LIN {X -0.158,Y -301.655,Z 469.672,A 0.000,B 0.000,C 90.000,E1 301.003} C_DIS
LIN {X -0.099,Y -317.062,Z 469.654,A 0.000,B 0.000,C 90.000,E1 297.719} C_DIS
LIN {X -0.042,Y -330.950,Z 469.640,A 0.000,B 0.000,C 90.000,E1 295.155} C_DIS
LIN {X 0.084,Y -344.129,Z 469.628,A 0.000,B 0.000,C 90.000,E1 292.950} C_DIS
LIN {X -0.112,Y -362.871,Z 469.612,A 0.000,B 0.000,C 90.000,E1 290.248} C_DIS
LIN {X -0.023,Y -381.291,Z 469.599,A 0.000,B 0.000,C 90.000,E1 287.873} C_DIS
LIN {X 0.019,Y -403.542,Z 469.585,A 0.000,B 0.000,C 90.000,E1 285.300} C_DIS
LIN {X 0.221,Y -426.591,Z 469.572,A 0.000,B 0.000,C 90.000,E1 282.883} C_DIS
LIN {X 0.019,Y -436.659,Z 469.566,A 0.000,B 0.000,C 90.000,E1 281.883} C_DIS
LIN {X 0.090,Y -446.267,Z 469.560,A 0.000,B 0.000,C 90.000,E1 280.838} C_DIS
LIN {X 0.109,Y -455.363,Z 469.554,A 0.000,B 0.000,C 90.000,E1 279.792} C_DIS
LIN {X 0.000,Y -461.575,Z 469.550,A 0.000,B 0.000,C 90.000,E1 279.029} C_DIS
LIN {X -0.130,Y -467.256,Z 469.546,A 0.000,B 0.000,C 90.000,E1 278.276} C_DIS
LIN {X 0.187,Y -472.386,Z 469.542,A 0.000,B 0.000,C 90.000,E1 277.473} C_DIS
LIN {X 0.155,Y -476.926,Z 469.537,A 0.000,B 0.000,C 90.000,E1 276.720} C_DIS
LIN {X 0.153,Y -480.963,Z 469.533,A 0.000,B 0.000,C 90.000,E1 275.967} C_DIS
LIN {X 0.136,Y -484.414,Z 469.529,A 0.000,B 0.000,C 90.000,E1 275.220} C_DIS
LIN {X 0.150,Y -487.205,Z 469.525,A 0.000,B 0.000,C 90.000,E1 274.473} C_DIS
LIN {X -0.144,Y -488.693,Z 469.522,A 0.000,B 0.000,C 90.000,E1 274.012} C_DIS
LIN {X 0.025,Y -489.834,Z 469.519,A 0.000,B 0.000,C 90.000,E1 273.498} C_DIS
LIN {X 0.235,Y -490.624,Z 469.517,A 0.000,B 0.000,C 90.000,E1 272.980} C_DIS
LIN {X -0.066,Y -491.068,Z 469.514,A 0.000,B 0.000,C 90.000,E1 272.522} C_DIS
LIN {X 0.131,Y -491.117,Z 469.511,A 0.000,B 0.000,C 90.000,E1 272.007} C_DIS
LIN {X -0.143,Y -490.735,Z 469.509,A 0.000,B 0.000,C 90.000,E1 271.547} C_DIS
LIN {X 0.057,Y -489.896,Z 469.506,A 0.000,B 0.000,C 90.000,E1 271.031} C_DIS
LIN {X -0.233,Y -488.534,Z 469.503,A 0.000,B 0.000,C 90.000,E1 270.573} C_DIS
LIN {X -0.038,Y -486.619,Z 469.500,A 0.000,B 0.000,C 90.000,E1 270.057} C_DIS
LIN {X 0.147,Y -484.034,Z 469.498,A 0.000,B 0.000,C 90.000,E1 269.542} C_DIS
LIN {X -0.168,Y -480.744,Z 469.495,A 0.000,B 0.000,C 90.000,E1 269.083} C_DIS
LIN {X -0.020,Y -476.512,Z 469.492,A 0.000,B 0.000,C 90.000,E1 268.568} C_DIS
LIN {X 0.119,Y -471.190,Z 469.489,A 0.000,B 0.000,C 90.000,E1 268.051} C_DIS
LIN {X 0.111,Y -465.151,Z 469.487,A 0.000,B 0.000,C 90.000,E1 267.593} C_DIS
LIN {X 0.111,Y -458.674,Z 469.484,A 0.000,B 0.000,C 90.000,E1 267.192} C_DIS
LIN {X 0.149,Y -452.078,Z 469.483,A 0.000,B 0.000,C 90.000,E1 266.849} C_DIS
LIN {X 0.109,Y -444.919,Z 469.481,A 0.000,B 0.000,C 90.000,E1 266.560} C_DIS
LIN {X 0.022,Y -437.347,Z 469.480,A 0.000,B 0.000,C 90.000,E1 266.331} C_DIS
LIN {X -0.069,Y -429.037,Z 469.479,A 0.000,B 0.000,C 90.000,E1 266.159} C_DIS
LIN {X -0.159,Y -419.638,Z 469.478,A 0.000,B 0.000,C 90.000,E1 266.045} C_DIS
LIN {X 0.136,Y -408.844,Z 469.477,A 0.000,B 0.000,C 90.000,E1 265.927} C_DIS
LIN {X 0.025,Y -180.917,Z 469.477,A 0.000,B 0.000,C 90.000,E1 265.927} C_DIS
LIN {X 0.054,Y -180.840,Z 469.472,A 0.000,B 0.000,C 90.000,E1 264.894} C_DIS
LIN {X -0.049,Y -178.880,Z 469.443,A 0.000,B 0.000,C 90.000,E1 259.690} C_DIS
LIN {X 0.027,Y -175.923,Z 469.414,A 0.000,B 0.000,C 90.000,E1 254.574} C_DIS
LIN {X -0.027,Y -175.360,Z 469.410,A 0.000,B 0.000,C 90.000,E1 253.740} C_DIS
LIN {X 0.031,Y -172.139,Z 469.386,A 0.000,B 0.000,C 90.000,E1 249.444} C_DIS
LIN {X 0.009,Y -171.602,Z 469.381,A 0.000,B 0.000,C 90.000,E1 248.592} C_DIS
LIN {X -0.003,Y -167.826,Z 469.357,A 0.000,B 0.000,C 90.000,E1 244.280} C_DIS
LIN {X 0.014,Y -166.550,Z 469.347,A 0.000,B 0.000,C 90.000,E1 242.538} C_DIS
LIN {X -0.074,Y -162.546,Z 469.323,A 0.000,B 0.000,C 90.000,E1 238.201} C_DIS
LIN {X -0.015,Y -161.223,Z 469.313,A 0.000,B 0.000,C 90.000,E1 236.421} C_DIS
LIN {X 0.021,Y -157.230,Z 469.289,A 0.000,B 0.000,C 90.000,E1 231.984} C_DIS
LIN {X 0.044,Y -155.955,Z 469.279,A 0.000,B 0.000,C 90.000,E1 230.194} C_DIS
LIN {X 0.002,Y -152.208,Z 469.254,A 0.000,B 0.000,C 90.000,E1 225.729} C_DIS
LIN {X 0.023,Y -150.452,Z 469.239,A 0.000,B 0.000,C 90.000,E1 223.014} C_DIS
LIN {X 0.050,Y -147.178,Z 469.214,A 0.000,B 0.000,C 90.000,E1 218.463} C_DIS
LIN {X 0.017,Y -145.195,Z 469.193,A 0.000,B 0.000,C 90.000,E1 214.818} C_DIS
LIN {X 0.051,Y -142.335,Z 469.163,A 0.000,B 0.000,C 90.000,E1 209.283} C_DIS
LIN {X -0.020,Y -141.724,Z 469.153,A 0.000,B 0.000,C 90.000,E1 207.462} C_DIS
LIN {X -0.038,Y -139.479,Z 469.116,A 0.000,B 0.000,C 90.000,E1 200.972} C_DIS
LIN {X -0.048,Y -138.976,Z 469.101,A 0.000,B 0.000,C 90.000,E1 198.181} C_DIS
LIN {X 0.073,Y -138.332,Z 469.054,A 0.000,B 0.000,C 90.000,E1 189.726} C_DIS
LIN {X -0.063,Y -139.432,Z 469.008,A 0.000,B 0.000,C 90.000,E1 181.375} C_DIS
LIN {X 0.017,Y -140.957,Z 468.976,A 0.000,B 0.000,C 90.000,E1 175.755} C_DIS
LIN {X -0.033,Y -142.713,Z 468.956,A 0.000,B 0.000,C 90.000,E1 172.064} C_DIS
LIN {X 0.067,Y -145.090,Z 468.930,A 0.000,B 0.000,C 90.000,E1 167.409} C_DIS
LIN {X 0.061,Y -147.714,Z 468.910,A 0.000,B 0.000,C 90.000,E1 163.740} C_DIS
LIN {X 0.003,Y -150.372,Z 468.890,A 0.000,B 0.000,C 90.000,E1 160.115} C_DIS
LIN {X 0.021,Y -153.799,Z 468.869,A 0.000,B 0.000,C 90.000,E1 156.485} C_DIS
LIN {X 0.081,Y -157.211,Z 468.849,A 0.000,B 0.000,C 90.000,E1 152.871} C_DIS
LIN {X 0.022,Y -161.376,Z 468.830,A 0.000,B 0.000,C 90.000,E1 149.331} C_DIS
LIN {X 0.033,Y -165.578,Z 468.810,A 0.000,B 0.000,C 90.000,E1 145.801} C_DIS
LIN {X 0.020,Y -170.497,Z 468.791,A 0.000,B 0.000,C 90.000,E1 142.316} C_DIS
LIN {X 0.065,Y -175.378,Z 468.772,A 0.000,B 0.000,C 90.000,E1 138.852} C_DIS
LIN {X -0.073,Y -181.002,Z 468.753,A 0.000,B 0.000,C 90.000,E1 135.486} C_DIS
LIN {X 0.051,Y -186.430,Z 468.734,A 0.000,B 0.000,C 90.000,E1 132.081} C_DIS
LIN {X 0.121,Y -191.056,Z 468.720,A 0.000,B 0.000,C 90.000,E1 129.564} C_DIS
LIN {X -0.048,Y -194.103,Z 468.710,A 0.000,B 0.000,C 90.000,E1 127.810} C_DIS
LIN {X -0.108,Y -291.699,Z 468.710,A 0.000,B 0.000,C 90.000,E1 127.810} C_DIS
LIN {X 0.063,Y -294.118,Z 468.710,A 0.000,B 0.000,C 90.000,E1 127.729} C_DIS
LIN {X -0.041,Y -299.359,Z 468.708,A 0.000,B 0.000,C 90.000,E1 127.443} C_DIS
LIN {X -0.149,Y -302.223,Z 468.706,A 0.000,B 0.000,C 90.000,E1 127.156} C_DIS
LIN {X 0.030,Y -304.266,Z 468.705,A 0.000,B 0.000,C 90.000,E1 126.824} C_DIS
LIN {X 0.149,Y -305.872,Z 468.703,A 0.000,B 0.000,C 90.000,E1 126.503} C_DIS
LIN {X -0.076,Y -307.278,Z 468.701,A 0.000,B 0.000,C 90.000,E1 126.217} C_DIS
LIN {X -0.055,Y -310.333,Z 468.696,A 0.000,B 0.000,C 90.000,E1 125.231} C_DIS
LIN {X -0.088,Y -320.951,Z 468.678,A 0.000,B 0.000,C 90.000,E1 122.005} C_DIS
LIN {X -0.112,Y -331.871,Z 468.662,A 0.000,B 0.000,C 90.000,E1 119.155} C_DIS
LIN {X -0.150,Y -344.193,Z 468.646,A 0.000,B 0.000,C 90.000,E1 116.360} C_DIS
LIN {X -0.016,Y -356.409,Z 468.633,A 0.000,B 0.000,C 90.000,E1 113.898} C_DIS
LIN {X -0.187,Y -369.906,Z 468.619,A 0.000,B 0.000,C 90.000,E1 111.535} C_DIS
LIN {X 0.190,Y -384.783,Z 468.607,A 0.000,B 0.000,C 90.000,E1 109.141} C_DIS
LIN {X -0.174,Y -401.147,Z 468.594,A 0.000,B 0.000,C 90.000,E1 106.913} C_DIS
LIN {X 0.022,Y -419.122,Z 468.581,A 0.000,B 0.000,C 90.000,E1 104.662} C_DIS
LIN {X -0.150,Y -438.706,Z 468.570,A 0.000,B 0.000,C 90.000,E1 102.535} C_DIS
LIN {X -0.130,Y -459.049,Z 468.559,A 0.000,B 0.000,C 90.000,E1 100.546} C_DIS
LIN {X -0.157,Y -482.472,Z 468.547,A 0.000,B 0.000,C 90.000,E1 98.511} C_DIS
LIN {X 0.005,Y -484.489,Z 468.546,A 0.000,B 0.000,C 90.000,E1 98.276} C_DIS
LIN {X -0.183,Y -486.247,Z 468.545,A 0.000,B 0.000,C 90.000,E1 98.049} C_DIS
LIN {X 0.181,Y -487.565,Z 468.543,A 0.000,B 0.000,C 90.000,E1 97.757} C_DIS
LIN {X -0.103,Y -489.207,Z 468.540,A 0.000,B 0.000,C 90.000,E1 97.296} C_DIS
LIN {X 0.106,Y -489.773,Z 468.538,A 0.000,B 0.000,C 90.000,E1 96.777} C_DIS
LIN {X -0.163,Y -489.358,Z 468.535,A 0.000,B 0.000,C 90.000,E1 96.315} C_DIS
LIN {X 0.059,Y -487.894,Z 468.532,A 0.000,B 0.000,C 90.000,E1 95.796} C_DIS
LIN {X -0.099,Y -486.692,Z 468.531,A 0.000,B 0.000,C 90.000,E1 95.568} C_DIS
LIN {X -0.209,Y -485.083,Z 468.530,A 0.000,B 0.000,C 90.000,E1 95.334} C_DIS
LIN {X -0.049,Y -475.019,Z 468.523,A 0.000,B 0.000,C 90.000,E1 94.073} C_DIS
LIN {X 0.111,Y -457.545,Z 468.510,A 0.000,B 0.000,C 90.000,E1 91.776} C_DIS
LIN {X -0.163,Y -445.267,Z 468.500,A 0.000,B 0.000,C 90.000,E1 90.000} C_DIS
LIN {X -0.208,Y -433.697,Z 468.490,A 0.000,B 0.000,C 90.000,E1 88.165} C_DIS
LIN {X 0.193,Y -419.113,Z 468.476,A 0.000,B 0.000,C 90.000,E1 85.698} C_DIS
LIN {X 0.149,Y -406.464,Z 468.464,A 0.000,B 0.000,C 90.000,E1 83.514} C_DIS
LIN {X -0.112,Y -395.623,Z 468.453,A 0.000,B 0.000,C 90.000,E1 81.602} C_DIS
LIN {X -0.159,Y -383.212,Z 468.441,A 0.000,B 0.000,C 90.000,E1 79.342} C_DIS
LIN {X 0.080,Y -369.445,Z 468.426,A 0.000,B 0.000,C 90.000,E1 76.700} C_DIS
LIN {X 0.029,Y -356.550,Z 468.411,A 0.000,B 0.000,C 90.000,E1 74.047} C_DIS
LIN {X 0.030,Y -345.025,Z 468.396,A 0.000,B 0.000,C 90.000,E1 71.329} C_DIS
LIN {X -0.159,Y -333.470,Z 468.379,A 0.000,B 0.000,C 90.000,E1 68.284} C_DIS
LIN {X 0.056,Y -324.572,Z 468.365,A 0.000,B 0.000,C 90.000,E1 65.741} C_DIS
LIN {X 0.091,Y -316.945,Z 468.353,A 0.000,B 0.000,C 90.000,E1 63.512} C_DIS
LIN {X -0.098,Y -308.433,Z 468.339,A 0.000,B 0.000,C 90.000,E1 60.973} C_DIS
LIN {X 0.074,Y -300.074,Z 468.324,A 0.000,B 0.000,C 90.000,E1 58.329} C_DIS
LIN {X 0.002,Y -290.135,Z 468.306,A 0.000,B 0.000,C 90.000,E1 55.022} C_DIS
LIN {X 0.033,Y -282.648,Z 468.291,A 0.000,B 0.000,C 90.000,E1 52.316} C_DIS
LIN {X -0.008,Y -276.960,Z 468.279,A 0.000,B 0.000,C 90.000,E1 50.275} C_DIS
LIN {X 0.010,Y -270.921,Z 468.268,A 0.000,B 0.000,C 90.000,E1 48.200} C_DIS
LIN {X -0.127,Y -264.601,Z 468.256,A 0.000,B 0.000,C 90.000,E1 46.134} C_DIS
LIN {X 0.179,Y -258.110,Z 468.244,A 0.000,B 0.000,C 90.000,E1 43.947} C_DIS
LIN {X 0.002,Y -251.544,Z 468.232,A 0.000,B 0.000,C 90.000,E1 41.838} C_DIS
LIN {X 0.090,Y -242.873,Z 468.216,A 0.000,B 0.000,C 90.000,E1 38.910} C_DIS
LIN {X 0.041,Y -234.668,Z 468.200,A 0.000,B 0.000,C 90.000,E1 35.964} C_DIS
LIN {X 0.033,Y -227.225,Z 468.183,A 0.000,B 0.000,C 90.000,E1 32.959} C_DIS
LIN {X -0.030,Y -220.513,Z 468.166,A 0.000,B 0.000,C 90.000,E1 29.922} C_DIS
LIN {X -0.007,Y -214.701,Z 468.149,A 0.000,B 0.000,C 90.000,E1 26.821} C_DIS
LIN {X 0.001,Y -208.464,Z 468.127,A 0.000,B 0.000,C 90.000,E1 22.898} C_DIS
LIN {X 0.067,Y -203.248,Z 468.105,A 0.000,B 0.000,C 90.000,E1 18.906} C_DIS
LIN {X 0.035,Y -199.029,Z 468.083,A 0.000,B 0.000,C 90.000,E1 14.898} C_DIS
LIN {X 0.082,Y -195.313,Z 468.056,A 0.000,B 0.000,C 90.000,E1 10.018} C_DIS
LIN {X 0.005,Y -192.428,Z 468.019,A 0.000,B 0.000,C 90.000,E1 3.498} C_DIS
LIN {X 0.027,Y -193.612,Z 467.956,A 0.000,B 0.000,C 90.000,E1 352.129} C_DIS
LIN {X 0.005,Y -196.608,Z 467.929,A 0.000,B 0.000,C 90.000,E1 347.229} C_DIS
LIN {X -0.008,Y -200.943,Z 467.902,A 0.000,B 0.000,C 90.000,E1 342.362} C_DIS
LIN {X 0.006,Y -205.588,Z 467.880,A 0.000,B 0.000,C 90.000,E1 338.337} C_DIS
LIN {X 0.009,Y -211.093,Z 467.858,A 0.000,B 0.000,C 90.000,E1 334.357} C_DIS
LIN {X 0.119,Y -216.069,Z 467.840,A 0.000,B 0.000,C 90.000,E1 331.179} C_DIS
LIN {X -0.017,Y -222.825,Z 467.818,A 0.000,B 0.000,C 90.000,E1 327.327} C_DIS
LIN {X -0.029,Y -230.159,Z 467.797,A 0.000,B 0.000,C 90.000,E1 323.497} C_DIS
LIN {X 0.053,Y -238.285,Z 467.776,A 0.000,B 0.000,C 90.000,E1 319.703} C_DIS
LIN {X -0.003,Y -245.579,Z 467.760,A 0.000,B 0.000,C 90.000,E1 316.743} C_DIS
LIN {X -0.036,Y -254.769,Z 467.741,A 0.000,B 0.000,C 90.000,E1 313.461} C_DIS
LIN {X -0.120,Y -265.095,Z 467.723,A 0.000,B 0.000,C 90.000,E1 310.253} C_DIS
LIN {X -0.037,Y -276.415,Z 467.706,A 0.000,B 0.000,C 90.000,E1 307.076} C_DIS
LIN {X -0.074,Y -288.634,Z 467.689,A 0.000,B 0.000,C 90.000,E1 303.992} C_DIS
LIN {X 0.173,Y -301.649,Z 467.672,A 0.000,B 0.000,C 90.000,E1 300.924} C_DIS
LIN {X -0.037,Y -317.088,Z 467.654,A 0.000,B 0.000,C 90.000,E1 297.692} C_DIS
LIN {X -0.065,Y -334.625,Z 467.636,A 0.000,B 0.000,C 90.000,E1 294.515} C_DIS
LIN {X -0.003,Y -346.171,Z 467.626,A 0.000,B 0.000,C 90.000,E1 292.642} C_DIS
LIN {X -0.208,Y -362.890,Z 467.612,A 0.000,B 0.000,C 90.000,E1 290.248} C_DIS
LIN {X -0.127,Y -383.715,Z 467.598,A 0.000,B 0.000,C 90.000,E1 287.583} C_DIS
LIN {X 0.056,Y -406.100,Z 467.583,A 0.000,B 0.000,C 90.000,E1 285.009} C_DIS
LIN {X 0.110,Y -426.722,Z 467.572,A 0.000,B 0.000,C 90.000,E1 282.883} C_DIS
LIN {X -0.120,Y -436.847,Z 467.566,A 0.000,B 0.000,C 90.000,E1 281.883} C_DIS
LIN {X -0.146,Y -446.582,Z 467.560,A 0.000,B 0.000,C 90.000,E1 280.838} C_DIS
LIN {X 0.116,Y -453.506,Z 467.556,A 0.000,B 0.000,C 90.000,E1 280.018} C_DIS
LIN {X 0.189,Y -461.868,Z 467.550,A 0.000,B 0.000,C 90.000,E1 278.973} C_DIS
LIN {X 0.065,Y -467.543,Z 467.546,A 0.000,B 0.000,C 90.000,E1 278.219} C_DIS
LIN {X -0.018,Y -472.658,Z 467.541,A 0.000,B 0.000,C 90.000,E1 277.466} C_DIS
LIN {X -0.111,Y -477.174,Z 467.537,A 0.000,B 0.000,C 90.000,E1 276.720} C_DIS
LIN {X -0.115,Y -481.179,Z 467.533,A 0.000,B 0.000,C 90.000,E1 275.967} C_DIS
LIN {X -0.130,Y -484.631,Z 467.529,A 0.000,B 0.000,C 90.000,E1 275.220} C_DIS
LIN {X -0.116,Y -487.443,Z 467.525,A 0.000,B 0.000,C 90.000,E1 274.473} C_DIS
LIN {X 0.077,Y -488.925,Z 467.522,A 0.000,B 0.000,C 90.000,E1 273.955} C_DIS
LIN {X -0.240,Y -490.031,Z 467.519,A 0.000,B 0.000,C 90.000,E1 273.498} C_DIS
LIN {X -0.029,Y -490.816,Z 467.517,A 0.000,B 0.000,C 90.000,E1 272.980} C_DIS
LIN {X 0.161,Y -491.229,Z 467.514,A 0.000,B 0.000,C 90.000,E1 272.465} C_DIS
LIN {X -0.131,Y -491.240,Z 467.511,A 0.000,B 0.000,C 90.000,E1 272.007} C_DIS
LIN {X 0.085,Y -490.808,Z 467.508,A 0.000,B 0.000,C 90.000,E1 271.489} C_DIS
LIN {X -0.203,Y -489.908,Z 467.506,A 0.000,B 0.000,C 90.000,E1 271.031} C_DIS
LIN {X -0.004,Y -488.535,Z 467.503,A 0.000,B 0.000,C 90.000,E1 270.516} C_DIS
LIN {X 0.190,Y -486.545,Z 467.500,A 0.000,B 0.000,C 90.000,E1 270.000} C_DIS
LIN {X -0.109,Y -483.920,Z 467.497,A 0.000,B 0.000,C 90.000,E1 269.542} C_DIS
LIN {X 0.057,Y -480.586,Z 467.495,A 0.000,B 0.000,C 90.000,E1 269.026} C_DIS
LIN {X 0.203,Y -476.308,Z 467.492,A 0.000,B 0.000,C 90.000,E1 268.511} C_DIS
LIN {X -0.133,Y -470.890,Z 467.489,A 0.000,B 0.000,C 90.000,E1 268.051} C_DIS
LIN {X -0.113,Y -464.803,Z 467.487,A 0.000,B 0.000,C 90.000,E1 267.593} C_DIS
LIN {X -0.072,Y -458.342,Z 467.484,A 0.000,B 0.000,C 90.000,E1 267.192} C_DIS
LIN {X 0.019,Y -451.643,Z 467.482,A 0.000,B 0.000,C 90.000,E1 266.846} C_DIS
LIN {X 0.058,Y -444.877,Z 467.481,A 0.000,B 0.000,C 90.000,E1 266.560} C_DIS
LIN {X -0.068,Y -437.009,Z 467.480,A 0.000,B 0.000,C 90.000,E1 266.331} C_DIS
LIN {X -0.150,Y -428.528,Z 467.479,A 0.000,B 0.000,C 90.000,E1 266.159} C_DIS
LIN {X -0.216,Y -418.896,Z 467.478,A 0.000,B 0.000,C 90.000,E1 266.045} C_DIS
LIN {X 0.111,Y -408.269,Z 467.477,A 0.000,B 0.000,C 90.000,E1 265.927} C_DIS
LIN {X 0.016,Y -180.917,Z 467.477,A 0.000,B 0.000,C 90.000,E1 265.927} C_DIS
LIN {X 0.047,Y -180.838,Z 467.472,A 0.000,B 0.000,C 90.000,E1 264.894} C_DIS
LIN {X -0.055,Y -178.879,Z 467.443,A 0.000,B 0.000,C 90.000,E1 259.690} C_DIS
LIN {X 0.020,Y -175.922,Z 467.414,A 0.000,B 0.000,C 90.000,E1 254.574} C_DIS
LIN {X -0.090,Y -174.620,Z 467.405,A 0.000,B 0.000,C 90.000,E1 252.906} C_DIS
LIN {X 0.002,Y -171.601,Z 467.381,A 0.000,B 0.000,C 90.000,E1 248.592} C_DIS
LIN {X -0.009,Y -167.823,Z 467.357,A 0.000,B 0.000,C 90.000,E1 244.280} C_DIS
LIN {X 0.008,Y -166.548,Z 467.347,A 0.000,B 0.000,C 90.000,E1 242.538} C_DIS
LIN {X -0.081,Y -162.544,Z 467.323,A 0.000,B 0.000,C 90.000,E1 238.201} C_DIS
LIN {X -0.021,Y -161.221,Z 467.313,A 0.000,B 0.000,C 90.000,E1 236.421} C_DIS
LIN {X 0.014,Y -157.228,Z 467.289,A 0.000,B 0.000,C 90.000,E1 231.984} C_DIS
LIN {X 0.037,Y -155.953,Z 467.279,A 0.000,B 0.000,C 90.000,E1 230.194} C_DIS
LIN {X -0.004,Y -152.206,Z 467.254,A 0.000,B 0.000,C 90.000,E1 225.729} C_DIS
LIN {X 0.016,Y -150.451,Z 467.239,A 0.000,B 0.000,C 90.000,E1 223.014} C_DIS
LIN {X 0.043,Y -147.177,Z 467.214,A 0.000,B 0.000,C 90.000,E1 218.463} C_DIS
LIN {X 0.010,Y -145.195,Z 467.193,A 0.000,B 0.000,C 90.000,E1 214.818} C_DIS
LIN {X 0.045,Y -142.334,Z 467.163,A 0.000,B 0.000,C 90.000,E1 209.283} C_DIS
LIN {X -0.026,Y -141.723,Z 467.152,A 0.000,B 0.000,C 90.000,E1 207.462} C_DIS
LIN {X -0.044,Y -139.478,Z 467.116,A 0.000,B 0.000,C 90.000,E1 200.972} C_DIS
LIN {X -0.055,Y -138.976,Z 467.101,A 0.000,B 0.000,C 90.000,E1 198.181} C_DIS
LIN {X 0.067,Y -138.332,Z 467.054,A 0.000,B 0.000,C 90.000,E1 189.726} C_DIS
LIN {X 0.070,Y -139.431,Z 467.007,A 0.000,B 0.000,C 90.000,E1 181.318} C_DIS
LIN {X 0.010,Y -140.958,Z 466.976,A 0.000,B 0.000,C 90.000,E1 175.755} C_DIS
LIN {X -0.040,Y -142.714,Z 466.956,A 0.000,B 0.000,C 90.000,E1 172.064} C_DIS
LIN {X 0.060,Y -145.091,Z 466.930,A 0.000,B 0.000,C 90.000,E1 167.409} C_DIS
LIN {X 0.056,Y -147.716,Z 466.910,A 0.000,B 0.000,C 90.000,E1 163.740} C_DIS
LIN {X -0.004,Y -150.373,Z 466.890,A 0.000,B 0.000,C 90.000,E1 160.115} C_DIS
LIN {X 0.014,Y -153.802,Z 466.869,A 0.000,B 0.000,C 90.000,E1 156.485} C_DIS
LIN {X 0.074,Y -157.213,Z 466.849,A 0.000,B 0.000,C 90.000,E1 152.871} C_DIS
LIN {X 0.015,Y -161.378,Z 466.830,A 0.000,B 0.000,C 90.000,E1 149.331} C_DIS
LIN {X 0.027,Y -165.581,Z 466.810,A 0.000,B 0.000,C 90.000,E1 145.801} C_DIS
LIN {X 0.013,Y -170.501,Z 466.791,A 0.000,B 0.000,C 90.000,E1 142.316} C_DIS
LIN {X 0.058,Y -175.381,Z 466.772,A 0.000,B 0.000,C 90.000,E1 138.852} C_DIS
LIN {X -0.080,Y -181.006,Z 466.753,A 0.000,B 0.000,C 90.000,E1 135.486} C_DIS
LIN {X 0.044,Y -186.434,Z 466.734,A 0.000,B 0.000,C 90.000,E1 132.081} C_DIS
LIN {X 0.113,Y -191.060,Z 466.720,A 0.000,B 0.000,C 90.000,E1 129.564} C_DIS
LIN {X 0.032,Y -194.204,Z 466.710,A 0.000,B 0.000,C 90.000,E1 127.729} C_DIS
LIN {X 0.014,Y -291.917,Z 466.710,A 0.000,B 0.000,C 90.000,E1 127.729} C_DIS
LIN {X 0.121,Y -294.651,Z 466.709,A 0.000,B 0.000,C 90.000,E1 127.649} C_DIS
LIN {X 0.010,Y -299.269,Z 466.708,A 0.000,B 0.000,C 90.000,E1 127.397} C_DIS
LIN {X -0.160,Y -301.942,Z 466.706,A 0.000,B 0.000,C 90.000,E1 127.156} C_DIS
LIN {X -0.180,Y -305.655,Z 466.703,A 0.000,B 0.000,C 90.000,E1 126.583} C_DIS
LIN {X 0.016,Y -307.140,Z 466.701,A 0.000,B 0.000,C 90.000,E1 126.217} C_DIS
LIN {X 0.034,Y -308.314,Z 466.699,A 0.000,B 0.000,C 90.000,E1 125.884} C_DIS
LIN {X 0.119,Y -318.630,Z 466.681,A 0.000,B 0.000,C 90.000,E1 122.625} C_DIS
LIN {X -0.083,Y -329.246,Z 466.665,A 0.000,B 0.000,C 90.000,E1 119.795} C_DIS
LIN {X 0.103,Y -341.240,Z 466.650,A 0.000,B 0.000,C 90.000,E1 116.950} C_DIS
LIN {X 0.036,Y -354.714,Z 466.635,A 0.000,B 0.000,C 90.000,E1 114.207} C_DIS
LIN {X -0.176,Y -368.038,Z 466.621,A 0.000,B 0.000,C 90.000,E1 111.844} C_DIS
LIN {X 0.153,Y -382.727,Z 466.608,A 0.000,B 0.000,C 90.000,E1 109.450} C_DIS
LIN {X 0.124,Y -398.891,Z 466.595,A 0.000,B 0.000,C 90.000,E1 107.166} C_DIS
LIN {X -0.008,Y -416.646,Z 466.583,A 0.000,B 0.000,C 90.000,E1 104.954} C_DIS
LIN {X 0.138,Y -436.049,Z 466.571,A 0.000,B 0.000,C 90.000,E1 102.771} C_DIS
LIN {X -0.010,Y -456.318,Z 466.560,A 0.000,B 0.000,C 90.000,E1 100.782} C_DIS
LIN {X 0.184,Y -477.118,Z 466.550,A 0.000,B 0.000,C 90.000,E1 98.916} C_DIS
LIN {X -0.077,Y -482.359,Z 466.547,A 0.000,B 0.000,C 90.000,E1 98.511} C_DIS
LIN {X 0.084,Y -484.444,Z 466.546,A 0.000,B 0.000,C 90.000,E1 98.276} C_DIS
LIN {X -0.103,Y -486.255,Z 466.545,A 0.000,B 0.000,C 90.000,E1 98.049} C_DIS
LIN {X -0.223,Y -487.615,Z 466.543,A 0.000,B 0.000,C 90.000,E1 97.814} C_DIS
LIN {X -0.024,Y -489.315,Z 466.541,A 0.000,B 0.000,C 90.000,E1 97.296} C_DIS
LIN {X 0.186,Y -489.931,Z 466.538,A 0.000,B 0.000,C 90.000,E1 96.777} C_DIS
LIN {X -0.083,Y -489.561,Z 466.535,A 0.000,B 0.000,C 90.000,E1 96.315} C_DIS
LIN {X 0.140,Y -488.153,Z 466.532,A 0.000,B 0.000,C 90.000,E1 95.796} C_DIS
LIN {X -0.018,Y -486.984,Z 466.531,A 0.000,B 0.000,C 90.000,E1 95.568} C_DIS
LIN {X -0.127,Y -485.420,Z 466.530,A 0.000,B 0.000,C 90.000,E1 95.334} C_DIS
LIN {X 0.036,Y -475.390,Z 466.523,A 0.000,B 0.000,C 90.000,E1 94.073} C_DIS
LIN {X -0.021,Y -456.050,Z 466.509,A 0.000,B 0.000,C 90.000,E1 91.547} C_DIS
LIN {X -0.123,Y -442.244,Z 466.497,A 0.000,B 0.000,C 90.000,E1 89.484} C_DIS
LIN {X 0.057,Y -427.435,Z 466.484,A 0.000,B 0.000,C 90.000,E1 87.078} C_DIS
LIN {X -0.116,Y -413.042,Z 466.470,A 0.000,B 0.000,C 90.000,E1 84.666} C_DIS
LIN {X 0.194,Y -400.568,Z 466.458,A 0.000,B 0.000,C 90.000,E1 82.413} C_DIS
LIN {X -0.178,Y -389.678,Z 466.447,A 0.000,B 0.000,C 90.000,E1 80.500} C_DIS
LIN {X 0.024,Y -380.432,Z 466.438,A 0.000,B 0.000,C 90.000,E1 78.757} C_DIS
LIN {X -0.189,Y -365.347,Z 466.421,A 0.000,B 0.000,C 90.000,E1 75.880} C_DIS
LIN {X -0.195,Y -354.196,Z 466.408,A 0.000,B 0.000,C 90.000,E1 73.504} C_DIS
LIN {X 0.080,Y -342.919,Z 466.393,A 0.000,B 0.000,C 90.000,E1 70.732} C_DIS
LIN {X -0.060,Y -331.475,Z 466.376,A 0.000,B 0.000,C 90.000,E1 67.667} C_DIS
LIN {X -0.109,Y -321.458,Z 466.360,A 0.000,B 0.000,C 90.000,E1 64.845} C_DIS
LIN {X -0.071,Y -312.772,Z 466.346,A 0.000,B 0.000,C 90.000,E1 62.281} C_DIS
LIN {X 0.060,Y -304.280,Z 466.332,A 0.000,B 0.000,C 90.000,E1 59.665} C_DIS
LIN {X 0.038,Y -294.052,Z 466.313,A 0.000,B 0.000,C 90.000,E1 56.373} C_DIS
LIN {X -0.127,Y -284.513,Z 466.295,A 0.000,B 0.000,C 90.000,E1 53.050} C_DIS
LIN {X 0.086,Y -278.881,Z 466.283,A 0.000,B 0.000,C 90.000,E1 50.964} C_DIS
LIN {X -0.069,Y -272.948,Z 466.272,A 0.000,B 0.000,C 90.000,E1 48.933} C_DIS
LIN {X 0.032,Y -266.721,Z 466.260,A 0.000,B 0.000,C 90.000,E1 46.824} C_DIS
LIN {X 0.010,Y -260.324,Z 466.248,A 0.000,B 0.000,C 90.000,E1 44.717} C_DIS
LIN {X -0.127,Y -253.782,Z 466.237,A 0.000,B 0.000,C 90.000,E1 42.609} C_DIS
LIN {X 0.000,Y -247.246,Z 466.225,A 0.000,B 0.000,C 90.000,E1 40.415} C_DIS
LIN {X -0.008,Y -236.714,Z 466.204,A 0.000,B 0.000,C 90.000,E1 36.744} C_DIS
LIN {X -0.152,Y -229.104,Z 466.188,A 0.000,B 0.000,C 90.000,E1 33.785} C_DIS
LIN {X -0.045,Y -222.146,Z 466.171,A 0.000,B 0.000,C 90.000,E1 30.718} C_DIS
LIN {X -0.073,Y -216.122,Z 466.153,A 0.000,B 0.000,C 90.000,E1 27.641} C_DIS
LIN {X -0.063,Y -210.880,Z 466.136,A 0.000,B 0.000,C 90.000,E1 24.515} C_DIS
LIN {X -0.039,Y -205.232,Z 466.114,A 0.000,B 0.000,C 90.000,E1 20.556} C_DIS
LIN {X -0.021,Y -200.601,Z 466.092,A 0.000,B 0.000,C 90.000,E1 16.551} C_DIS
LIN {X -0.100,Y -196.945,Z 466.069,A 0.000,B 0.000,C 90.000,E1 12.535} C_DIS
LIN {X 0.084,Y -193.512,Z 466.038,A 0.000,B 0.000,C 90.000,E1 6.777} C_DIS
LIN {X 0.080,Y -193.113,Z 465.961,A 0.000,B 0.000,C 90.000,E1 352.932} C_DIS
LIN {X -0.006,Y -196.481,Z 465.929,A 0.000,B 0.000,C 90.000,E1 347.229} C_DIS
LIN {X -0.025,Y -200.783,Z 465.902,A 0.000,B 0.000,C 90.000,E1 342.362} C_DIS
LIN {X -0.017,Y -205.404,Z 465.880,A 0.000,B 0.000,C 90.000,E1 338.337} C_DIS
LIN {X 0.071,Y -210.921,Z 465.858,A 0.000,B 0.000,C 90.000,E1 334.332} C_DIS
LIN {X 0.030,Y -217.220,Z 465.836,A 0.000,B 0.000,C 90.000,E1 330.411} C_DIS
LIN {X -0.058,Y -222.680,Z 465.818,A 0.000,B 0.000,C 90.000,E1 327.327} C_DIS
LIN {X -0.075,Y -229.999,Z 465.797,A 0.000,B 0.000,C 90.000,E1 323.497} C_DIS
LIN {X 0.000,Y -238.139,Z 465.776,A 0.000,B 0.000,C 90.000,E1 319.703} C_DIS
LIN {X 0.084,Y -247.370,Z 465.756,A 0.000,B 0.000,C 90.000,E1 315.972} C_DIS
LIN {X 0.122,Y -256.853,Z 465.737,A 0.000,B 0.000,C 90.000,E1 312.690} C_DIS
LIN {X 0.105,Y -267.433,Z 465.719,A 0.000,B 0.000,C 90.000,E1 309.483} C_DIS
LIN {X -0.078,Y -279.034,Z 465.702,A 0.000,B 0.000,C 90.000,E1 306.377} C_DIS
LIN {X -0.055,Y -292.877,Z 465.683,A 0.000,B 0.000,C 90.000,E1 302.959} C_DIS
LIN {X 0.000,Y -306.143,Z 465.666,A 0.000,B 0.000,C 90.000,E1 299.951} C_DIS
LIN {X 0.146,Y -320.455,Z 465.650,A 0.000,B 0.000,C 90.000,E1 297.001} C_DIS
LIN {X -0.063,Y -338.348,Z 465.633,A 0.000,B 0.000,C 90.000,E1 293.875} C_DIS
LIN {X 0.018,Y -356.478,Z 465.617,A 0.000,B 0.000,C 90.000,E1 291.099} C_DIS
LIN {X -0.101,Y -369.646,Z 465.607,A 0.000,B 0.000,C 90.000,E1 289.322} C_DIS
LIN {X 0.095,Y -393.537,Z 465.591,A 0.000,B 0.000,C 90.000,E1 286.386} C_DIS
LIN {X -0.102,Y -416.450,Z 465.577,A 0.000,B 0.000,C 90.000,E1 283.939} C_DIS
LIN {X 0.189,Y -431.864,Z 465.569,A 0.000,B 0.000,C 90.000,E1 282.355} C_DIS
LIN {X -0.156,Y -441.778,Z 465.563,A 0.000,B 0.000,C 90.000,E1 281.366} C_DIS
LIN {X -0.109,Y -451.273,Z 465.557,A 0.000,B 0.000,C 90.000,E1 280.310} C_DIS
LIN {X -0.065,Y -459.852,Z 465.551,A 0.000,B 0.000,C 90.000,E1 279.265} C_DIS
LIN {X -0.213,Y -465.749,Z 465.547,A 0.000,B 0.000,C 90.000,E1 278.511} C_DIS
LIN {X 0.159,Y -471.043,Z 465.543,A 0.000,B 0.000,C 90.000,E1 277.701} C_DIS
LIN {X 0.107,Y -475.760,Z 465.539,A 0.000,B 0.000,C 90.000,E1 276.947} C_DIS
LIN {X 0.044,Y -479.960,Z 465.534,A 0.000,B 0.000,C 90.000,E1 276.201} C_DIS
LIN {X 0.019,Y -483.618,Z 465.530,A 0.000,B 0.000,C 90.000,E1 275.454} C_DIS
LIN {X 0.197,Y -485.745,Z 465.528,A 0.000,B 0.000,C 90.000,E1 274.935} C_DIS
LIN {X -0.097,Y -487.565,Z 465.525,A 0.000,B 0.000,C 90.000,E1 274.473} C_DIS
LIN {X 0.098,Y -489.058,Z 465.522,A 0.000,B 0.000,C 90.000,E1 273.955} C_DIS
LIN {X -0.219,Y -490.199,Z 465.519,A 0.000,B 0.000,C 90.000,E1 273.498} C_DIS
LIN {X -0.008,Y -490.973,Z 465.517,A 0.000,B 0.000,C 90.000,E1 272.980} C_DIS
LIN {X 0.185,Y -491.371,Z 465.514,A 0.000,B 0.000,C 90.000,E1 272.465} C_DIS
LIN {X -0.107,Y -491.331,Z 465.511,A 0.000,B 0.000,C 90.000,E1 272.007} C_DIS
LIN {X 0.110,Y -490.932,Z 465.508,A 0.000,B 0.000,C 90.000,E1 271.489} C_DIS
LIN {X -0.178,Y -490.012,Z 465.506,A 0.000,B 0.000,C 90.000,E1 271.031} C_DIS
LIN {X 0.023,Y -488.622,Z 465.503,A 0.000,B 0.000,C 90.000,E1 270.516} C_DIS
LIN {X 0.217,Y -486.643,Z 465.500,A 0.000,B 0.000,C 90.000,E1 270.000} C_DIS
LIN {X -0.083,Y -484.046,Z 465.497,A 0.000,B 0.000,C 90.000,E1 269.542} C_DIS
LIN {X -0.240,Y -482.489,Z 465.496,A 0.000,B 0.000,C 90.000,E1 269.312} C_DIS
LIN {X -0.082,Y -478.649,Z 465.493,A 0.000,B 0.000,C 90.000,E1 268.797} C_DIS
LIN {X 0.231,Y -476.420,Z 465.492,A 0.000,B 0.000,C 90.000,E1 268.511} C_DIS
LIN {X -0.105,Y -471.016,Z 465.489,A 0.000,B 0.000,C 90.000,E1 268.051} C_DIS
LIN {X -0.100,Y -464.953,Z 465.487,A 0.000,B 0.000,C 90.000,E1 267.593} C_DIS
LIN {X -0.071,Y -458.484,Z 465.484,A 0.000,B 0.000,C 90.000,E1 267.192} C_DIS
LIN {X -0.021,Y -451.645,Z 465.482,A 0.000,B 0.000,C 90.000,E1 266.846} C_DIS
LIN {X 0.012,Y -444.807,Z 465.481,A 0.000,B 0.000,C 90.000,E1 266.560} C_DIS
LIN {X -0.088,Y -437.088,Z 465.480,A 0.000,B 0.000,C 90.000,E1 266.331} C_DIS
LIN {X -0.166,Y -428.532,Z 465.479,A 0.000,B 0.000,C 90.000,E1 266.159} C_DIS
LIN {X 0.187,Y -418.720,Z 465.478,A 0.000,B 0.000,C 90.000,E1 265.988} C_DIS
LIN {X 0.104,Y -407.968,Z 465.477,A 0.000,B 0.000,C 90.000,E1 265.927} C_DIS
LIN {X 0.013,Y -180.917,Z 465.477,A 0.000,B 0.000,C 90.000,E1 265.927} C_DIS
LIN {X 0.045,Y -180.839,Z 465.472,A 0.000,B 0.000,C 90.000,E1 264.894} C_DIS
LIN {X -0.058,Y -178.879,Z 465.443,A 0.000,B 0.000,C 90.000,E1 259.690} C_DIS
LIN {X 0.018,Y -175.922,Z 465.414,A 0.000,B 0.000,C 90.000,E1 254.574} C_DIS
LIN {X -0.093,Y -174.619,Z 465.405,A 0.000,B 0.000,C 90.000,E1 252.906} C_DIS
LIN {X 0.000,Y -171.600,Z 465.381,A 0.000,B 0.000,C 90.000,E1 248.592} C_DIS
LIN {X -0.012,Y -167.823,Z 465.357,A 0.000,B 0.000,C 90.000,E1 244.280} C_DIS
LIN {X 0.006,Y -166.547,Z 465.347,A 0.000,B 0.000,C 90.000,E1 242.538} C_DIS
LIN {X -0.083,Y -162.543,Z 465.323,A 0.000,B 0.000,C 90.000,E1 238.201} C_DIS
LIN {X -0.023,Y -161.221,Z 465.313,A 0.000,B 0.000,C 90.000,E1 236.421} C_DIS
LIN {X 0.012,Y -157.227,Z 465.289,A 0.000,B 0.000,C 90.000,E1 231.984} C_DIS
LIN {X 0.035,Y -155.952,Z 465.279,A 0.000,B 0.000,C 90.000,E1 230.194} C_DIS
LIN {X -0.006,Y -152.205,Z 465.254,A 0.000,B 0.000,C 90.000,E1 225.729} C_DIS
LIN {X 0.015,Y -150.451,Z 465.239,A 0.000,B 0.000,C 90.000,E1 223.014} C_DIS
LIN {X 0.041,Y -147.176,Z 465.214,A 0.000,B 0.000,C 90.000,E1 218.463} C_DIS
LIN {X 0.009,Y -145.193,Z 465.193,A 0.000,B 0.000,C 90.000,E1 214.818} C_DIS
LIN {X 0.043,Y -142.334,Z 465.163,A 0.000,B 0.000,C 90.000,E1 209.283} C_DIS
LIN {X -0.028,Y -141.723,Z 465.152,A 0.000,B 0.000,C 90.000,E1 207.462} C_DIS
LIN {X -0.045,Y -139.478,Z 465.116,A 0.000,B 0.000,C 90.000,E1 200.972} C_DIS
LIN {X -0.057,Y -138.976,Z 465.101,A 0.000,B 0.000,C 90.000,E1 198.181} C_DIS
LIN {X 0.065,Y -138.331,Z 465.054,A 0.000,B 0.000,C 90.000,E1 189.726} C_DIS
LIN {X 0.068,Y -139.431,Z 465.007,A 0.000,B 0.000,C 90.000,E1 181.318} C_DIS
LIN {X 0.008,Y -140.958,Z 464.976,A 0.000,B 0.000,C 90.000,E1 175.755} C_DIS
LIN {X -0.042,Y -142.714,Z 464.956,A 0.000,B 0.000,C 90.000,E1 172.064} C_DIS
LIN {X 0.058,Y -145.092,Z 464.930,A 0.000,B 0.000,C 90.000,E1 167.409} C_DIS
LIN {X 0.054,Y -147.717,Z 464.910,A 0.000,B 0.000,C 90.000,E1 163.740} C_DIS
LIN {X -0.006,Y -150.374,Z 464.890,A 0.000,B 0.000,C 90.000,E1 160.115} C_DIS
LIN {X 0.013,Y -153.803,Z 464.869,A 0.000,B 0.000,C 90.000,E1 156.485} C_DIS
LIN {X 0.072,Y -157.214,Z 464.849,A 0.000,B 0.000,C 90.000,E1 152.871} C_DIS
LIN {X 0.013,Y -161.380,Z 464.830,A 0.000,B 0.000,C 90.000,E1 149.331} C_DIS
LIN {X 0.024,Y -165.582,Z 464.810,A 0.000,B 0.000,C 90.000,E1 145.801} C_DIS
LIN {X 0.010,Y -170.502,Z 464.791,A 0.000,B 0.000,C 90.000,E1 142.316} C_DIS
LIN {X 0.055,Y -175.383,Z 464.771,A 0.000,B 0.000,C 90.000,E1 138.852} C_DIS
LIN {X -0.082,Y -181.007,Z 464.753,A 0.000,B 0.000,C 90.000,E1 135.486} C_DIS
LIN {X 0.042,Y -186.435,Z 464.734,A 0.000,B 0.000,C 90.000,E1 132.081} C_DIS
LIN {X 0.111,Y -191.061,Z 464.720,A 0.000,B 0.000,C 90.000,E1 129.564} C_DIS
LIN {X 0.023,Y -194.290,Z 464.709,A 0.000,B 0.000,C 90.000,E1 127.684} C_DIS
LIN {X -0.015,Y -291.952,Z 464.709,A 0.000,B 0.000,C 90.000,E1 127.684} C_DIS
LIN {X 0.114,Y -292.785,Z 464.709,A 0.000,B 0.000,C 90.000,E1 127.649} C_DIS
LIN {X 0.005,Y -298.761,Z 464.708,A 0.000,B 0.000,C 90.000,E1 127.397} C_DIS
LIN {X -0.164,Y -301.629,Z 464.706,A 0.000,B 0.000,C 90.000,E1 127.156} C_DIS
LIN {X -0.018,Y -305.348,Z 464.703,A 0.000,B 0.000,C 90.000,E1 126.583} C_DIS
LIN {X -0.003,Y -306.929,Z 464.701,A 0.000,B 0.000,C 90.000,E1 126.251} C_DIS
LIN {X -0.055,Y -308.179,Z 464.700,A 0.000,B 0.000,C 90.000,E1 125.931} C_DIS
LIN {X 0.086,Y -319.620,Z 464.680,A 0.000,B 0.000,C 90.000,E1 122.339} C_DIS
LIN {X 0.024,Y -330.373,Z 464.664,A 0.000,B 0.000,C 90.000,E1 119.489} C_DIS
LIN {X -0.043,Y -342.509,Z 464.648,A 0.000,B 0.000,C 90.000,E1 116.693} C_DIS
LIN {X -0.086,Y -356.143,Z 464.633,A 0.000,B 0.000,C 90.000,E1 113.951} C_DIS
LIN {X 0.073,Y -369.617,Z 464.620,A 0.000,B 0.000,C 90.000,E1 111.535} C_DIS
LIN {X -0.038,Y -384.469,Z 464.607,A 0.000,B 0.000,C 90.000,E1 109.214} C_DIS
LIN {X 0.091,Y -400.807,Z 464.594,A 0.000,B 0.000,C 90.000,E1 106.913} C_DIS
LIN {X -0.115,Y -418.752,Z 464.582,A 0.000,B 0.000,C 90.000,E1 104.717} C_DIS
LIN {X 0.114,Y -438.316,Z 464.570,A 0.000,B 0.000,C 90.000,E1 102.535} C_DIS
LIN {X 0.121,Y -458.650,Z 464.559,A 0.000,B 0.000,C 90.000,E1 100.546} C_DIS
LIN {X 0.080,Y -482.125,Z 464.547,A 0.000,B 0.000,C 90.000,E1 98.511} C_DIS
LIN {X 0.241,Y -484.310,Z 464.546,A 0.000,B 0.000,C 90.000,E1 98.276} C_DIS
LIN {X 0.105,Y -486.155,Z 464.545,A 0.000,B 0.000,C 90.000,E1 98.049} C_DIS
LIN {X 0.037,Y -487.549,Z 464.543,A 0.000,B 0.000,C 90.000,E1 97.814} C_DIS
LIN {X 0.236,Y -489.362,Z 464.541,A 0.000,B 0.000,C 90.000,E1 97.296} C_DIS
LIN {X -0.041,Y -490.070,Z 464.538,A 0.000,B 0.000,C 90.000,E1 96.834} C_DIS
LIN {X 0.178,Y -489.791,Z 464.535,A 0.000,B 0.000,C 90.000,E1 96.315} C_DIS
LIN {X -0.086,Y -488.485,Z 464.532,A 0.000,B 0.000,C 90.000,E1 95.853} C_DIS
LIN {X -0.242,Y -487.380,Z 464.531,A 0.000,B 0.000,C 90.000,E1 95.625} C_DIS
LIN {X 0.133,Y -485.896,Z 464.530,A 0.000,B 0.000,C 90.000,E1 95.334} C_DIS
LIN {X -0.002,Y -477.985,Z 464.524,A 0.000,B 0.000,C 90.000,E1 94.359} C_DIS
LIN {X -0.005,Y -458.402,Z 464.510,A 0.000,B 0.000,C 90.000,E1 91.835} C_DIS
LIN {X 0.200,Y -446.025,Z 464.500,A 0.000,B 0.000,C 90.000,E1 90.000} C_DIS
LIN {X -0.116,Y -432.740,Z 464.488,A 0.000,B 0.000,C 90.000,E1 87.936} C_DIS
LIN {X -0.160,Y -418.208,Z 464.475,A 0.000,B 0.000,C 90.000,E1 85.527} C_DIS
LIN {X -0.120,Y -404.092,Z 464.461,A 0.000,B 0.000,C 90.000,E1 83.053} C_DIS
LIN {X -0.032,Y -393.230,Z 464.450,A 0.000,B 0.000,C 90.000,E1 81.084} C_DIS
LIN {X -0.110,Y -382.444,Z 464.439,A 0.000,B 0.000,C 90.000,E1 79.106} C_DIS
LIN {X 0.102,Y -367.262,Z 464.423,A 0.000,B 0.000,C 90.000,E1 76.172} C_DIS
LIN {X 0.136,Y -355.964,Z 464.410,A 0.000,B 0.000,C 90.000,E1 73.795} C_DIS
LIN {X 0.024,Y -344.501,Z 464.395,A 0.000,B 0.000,C 90.000,E1 71.094} C_DIS
LIN {X -0.064,Y -332.916,Z 464.378,A 0.000,B 0.000,C 90.000,E1 68.028} C_DIS
LIN {X 0.136,Y -323.925,Z 464.364,A 0.000,B 0.000,C 90.000,E1 65.485} C_DIS
LIN {X 0.076,Y -315.172,Z 464.350,A 0.000,B 0.000,C 90.000,E1 62.948} C_DIS
LIN {X -0.026,Y -306.578,Z 464.335,A 0.000,B 0.000,C 90.000,E1 60.383} C_DIS
LIN {X -0.125,Y -296.182,Z 464.317,A 0.000,B 0.000,C 90.000,E1 57.120} C_DIS
LIN {X 0.015,Y -286.475,Z 464.299,A 0.000,B 0.000,C 90.000,E1 53.749} C_DIS
LIN {X 0.095,Y -280.864,Z 464.287,A 0.000,B 0.000,C 90.000,E1 51.698} C_DIS
LIN {X -0.024,Y -275.032,Z 464.276,A 0.000,B 0.000,C 90.000,E1 49.666} C_DIS
LIN {X 0.138,Y -268.910,Z 464.264,A 0.000,B 0.000,C 90.000,E1 47.553} C_DIS
LIN {X -0.034,Y -262.614,Z 464.253,A 0.000,B 0.000,C 90.000,E1 45.486} C_DIS
LIN {X 0.053,Y -256.120,Z 464.241,A 0.000,B 0.000,C 90.000,E1 43.338} C_DIS
LIN {X -0.153,Y -249.593,Z 464.229,A 0.000,B 0.000,C 90.000,E1 41.229} C_DIS
LIN {X 0.063,Y -238.917,Z 464.209,A 0.000,B 0.000,C 90.000,E1 37.523} C_DIS
LIN {X 0.101,Y -231.073,Z 464.192,A 0.000,B 0.000,C 90.000,E1 34.532} C_DIS
LIN {X -0.060,Y -223.930,Z 464.175,A 0.000,B 0.000,C 90.000,E1 31.544} C_DIS
LIN {X 0.069,Y -217.631,Z 464.158,A 0.000,B 0.000,C 90.000,E1 28.437} C_DIS
LIN {X 0.022,Y -212.219,Z 464.141,A 0.000,B 0.000,C 90.000,E1 25.335} C_DIS
LIN {X -0.032,Y -206.343,Z 464.119,A 0.000,B 0.000,C 90.000,E1 21.408} C_DIS
LIN {X 0.022,Y -201.480,Z 464.097,A 0.000,B 0.000,C 90.000,E1 17.402} C_DIS
LIN {X 0.074,Y -197.604,Z 464.074,A 0.000,B 0.000,C 90.000,E1 13.355} C_DIS
LIN {X -0.050,Y -194.288,Z 464.047,A 0.000,B 0.000,C 90.000,E1 8.511} C_DIS
LIN {X -0.030,Y -191.907,Z 464.011,A 0.000,B 0.000,C 90.000,E1 1.949} C_DIS
LIN {X 0.014,Y -193.359,Z 463.956,A 0.000,B 0.000,C 90.000,E1 352.129} C_DIS
LIN {X -0.018,Y -196.344,Z 463.929,A 0.000,B 0.000,C 90.000,E1 347.229} C_DIS
LIN {X 0.063,Y -199.825,Z 463.906,A 0.000,B 0.000,C 90.000,E1 343.142} C_DIS
LIN {X -0.027,Y -204.225,Z 463.884,A 0.000,B 0.000,C 90.000,E1 339.135} C_DIS
LIN {X -0.060,Y -209.574,Z 463.862,A 0.000,B 0.000,C 90.000,E1 335.153} C_DIS
LIN {X 0.051,Y -215.741,Z 463.840,A 0.000,B 0.000,C 90.000,E1 331.179} C_DIS
LIN {X 0.007,Y -221.136,Z 463.823,A 0.000,B 0.000,C 90.000,E1 328.074} C_DIS
LIN {X 0.132,Y -228.335,Z 463.801,A 0.000,B 0.000,C 90.000,E1 324.196} C_DIS
LIN {X 0.017,Y -236.269,Z 463.780,A 0.000,B 0.000,C 90.000,E1 320.436} C_DIS
LIN {X 0.059,Y -245.287,Z 463.760,A 0.000,B 0.000,C 90.000,E1 316.701} C_DIS
LIN {X 0.026,Y -254.523,Z 463.741,A 0.000,B 0.000,C 90.000,E1 313.419} C_DIS
LIN {X 0.120,Y -264.911,Z 463.723,A 0.000,B 0.000,C 90.000,E1 310.172} C_DIS
LIN {X 0.038,Y -276.307,Z 463.706,A 0.000,B 0.000,C 90.000,E1 307.030} C_DIS
LIN {X 0.044,Y -287.168,Z 463.690,A 0.000,B 0.000,C 90.000,E1 304.278} C_DIS
LIN {X -0.001,Y -300.170,Z 463.674,A 0.000,B 0.000,C 90.000,E1 301.258} C_DIS
LIN {X 0.013,Y -315.546,Z 463.655,A 0.000,B 0.000,C 90.000,E1 297.975} C_DIS
LIN {X -0.004,Y -325.701,Z 463.645,A 0.000,B 0.000,C 90.000,E1 296.052} C_DIS
LIN {X 0.132,Y -342.225,Z 463.629,A 0.000,B 0.000,C 90.000,E1 293.206} C_DIS
LIN {X 0.069,Y -362.928,Z 463.612,A 0.000,B 0.000,C 90.000,E1 290.174} C_DIS
LIN {X -0.187,Y -386.207,Z 463.596,A 0.000,B 0.000,C 90.000,E1 287.275} C_DIS
LIN {X -0.068,Y -406.081,Z 463.583,A 0.000,B 0.000,C 90.000,E1 285.009} C_DIS
LIN {X -0.072,Y -426.388,Z 463.572,A 0.000,B 0.000,C 90.000,E1 282.939} C_DIS
LIN {X 0.067,Y -436.511,Z 463.566,A 0.000,B 0.000,C 90.000,E1 281.895} C_DIS
LIN {X 0.156,Y -446.287,Z 463.560,A 0.000,B 0.000,C 90.000,E1 280.838} C_DIS
LIN {X -0.027,Y -453.225,Z 463.556,A 0.000,B 0.000,C 90.000,E1 280.074} C_DIS
LIN {X 0.040,Y -461.635,Z 463.550,A 0.000,B 0.000,C 90.000,E1 279.029} C_DIS
LIN {X -0.089,Y -467.364,Z 463.546,A 0.000,B 0.000,C 90.000,E1 278.276} C_DIS
LIN {X -0.239,Y -472.504,Z 463.542,A 0.000,B 0.000,C 90.000,E1 277.530} C_DIS
LIN {X 0.200,Y -477.056,Z 463.537,A 0.000,B 0.000,C 90.000,E1 276.720} C_DIS
LIN {X 0.198,Y -481.115,Z 463.533,A 0.000,B 0.000,C 90.000,E1 275.967} C_DIS
LIN {X 0.184,Y -484.683,Z 463.529,A 0.000,B 0.000,C 90.000,E1 275.220} C_DIS
LIN {X 0.200,Y -487.583,Z 463.525,A 0.000,B 0.000,C 90.000,E1 274.473} C_DIS
LIN {X -0.092,Y -489.110,Z 463.522,A 0.000,B 0.000,C 90.000,E1 274.012} C_DIS
LIN {X 0.079,Y -490.290,Z 463.519,A 0.000,B 0.000,C 90.000,E1 273.498} C_DIS
LIN {X -0.199,Y -491.079,Z 463.517,A 0.000,B 0.000,C 90.000,E1 273.037} C_DIS
LIN {X -0.007,Y -491.501,Z 463.514,A 0.000,B 0.000,C 90.000,E1 272.522} C_DIS
LIN {X 0.193,Y -491.460,Z 463.511,A 0.000,B 0.000,C 90.000,E1 272.007} C_DIS
LIN {X -0.079,Y -491.084,Z 463.509,A 0.000,B 0.000,C 90.000,E1 271.547} C_DIS
LIN {X 0.122,Y -490.175,Z 463.506,A 0.000,B 0.000,C 90.000,E1 271.031} C_DIS
LIN {X -0.166,Y -488.804,Z 463.503,A 0.000,B 0.000,C 90.000,E1 270.573} C_DIS
LIN {X 0.031,Y -486.898,Z 463.500,A 0.000,B 0.000,C 90.000,E1 270.057} C_DIS
LIN {X 0.218,Y -484.347,Z 463.498,A 0.000,B 0.000,C 90.000,E1 269.542} C_DIS
LIN {X -0.097,Y -481.063,Z 463.495,A 0.000,B 0.000,C 90.000,E1 269.083} C_DIS
LIN {X 0.053,Y -476.822,Z 463.492,A 0.000,B 0.000,C 90.000,E1 268.568} C_DIS
LIN {X 0.192,Y -471.543,Z 463.489,A 0.000,B 0.000,C 90.000,E1 268.051} C_DIS
LIN {X 0.162,Y -465.574,Z 463.487,A 0.000,B 0.000,C 90.000,E1 267.593} C_DIS
LIN {X 0.091,Y -458.949,Z 463.484,A 0.000,B 0.000,C 90.000,E1 267.192} C_DIS
LIN {X 0.124,Y -452.271,Z 463.483,A 0.000,B 0.000,C 90.000,E1 266.849} C_DIS
LIN {X 0.129,Y -445.261,Z 463.481,A 0.000,B 0.000,C 90.000,E1 266.560} C_DIS
LIN {X 0.029,Y -437.817,Z 463.480,A 0.000,B 0.000,C 90.000,E1 266.331} C_DIS
LIN {X -0.058,Y -429.417,Z 463.479,A 0.000,B 0.000,C 90.000,E1 266.159} C_DIS
LIN {X -0.136,Y -420.085,Z 463.478,A 0.000,B 0.000,C 90.000,E1 266.045} C_DIS
LIN {X 0.101,Y -407.405,Z 463.477,A 0.000,B 0.000,C 90.000,E1 265.927} C_DIS
LIN {X 0.022,Y -180.917,Z 463.477,A 0.000,B 0.000,C 90.000,E1 265.927} C_DIS
LIN {X -0.075,Y -180.871,Z 463.472,A 0.000,B 0.000,C 90.000,E1 265.065} C_DIS
LIN {X -0.018,Y -178.986,Z 463.444,A 0.000,B 0.000,C 90.000,E1 259.982} C_DIS
LIN {X -0.007,Y -177.966,Z 463.435,A 0.000,B 0.000,C 90.000,E1 258.285} C_DIS
LIN {X 0.012,Y -175.608,Z 463.411,A 0.000,B 0.000,C 90.000,E1 254.031} C_DIS
LIN {X 0.024,Y -172.332,Z 463.388,A 0.000,B 0.000,C 90.000,E1 249.752} C_DIS
LIN {X 0.003,Y -171.808,Z 463.383,A 0.000,B 0.000,C 90.000,E1 248.901} C_DIS
LIN {X 0.011,Y -170.269,Z 463.373,A 0.000,B 0.000,C 90.000,E1 247.177} C_DIS
LIN {X -0.053,Y -166.811,Z 463.349,A 0.000,B 0.000,C 90.000,E1 242.871} C_DIS
LIN {X 0.004,Y -162.793,Z 463.325,A 0.000,B 0.000,C 90.000,E1 238.486} C_DIS
LIN {X 0.064,Y -161.481,Z 463.315,A 0.000,B 0.000,C 90.000,E1 236.707} C_DIS
LIN {X -0.020,Y -157.477,Z 463.291,A 0.000,B 0.000,C 90.000,E1 232.316} C_DIS
LIN {X 0.037,Y -155.492,Z 463.276,A 0.000,B 0.000,C 90.000,E1 229.622} C_DIS
LIN {X -0.031,Y -151.798,Z 463.251,A 0.000,B 0.000,C 90.000,E1 225.162} C_DIS
LIN {X -0.017,Y -150.007,Z 463.236,A 0.000,B 0.000,C 90.000,E1 222.447} C_DIS
LIN {X 0.014,Y -146.834,Z 463.211,A 0.000,B 0.000,C 90.000,E1 217.890} C_DIS
LIN {X 0.000,Y -145.415,Z 463.195,A 0.000,B 0.000,C 90.000,E1 215.152} C_DIS
LIN {X 0.036,Y -142.844,Z 463.170,A 0.000,B 0.000,C 90.000,E1 210.541} C_DIS
LIN {X -0.035,Y -141.458,Z 463.149,A 0.000,B 0.000,C 90.000,E1 206.873} C_DIS
LIN {X 0.005,Y -139.374,Z 463.113,A 0.000,B 0.000,C 90.000,E1 200.355} C_DIS
LIN {X -0.053,Y -138.824,Z 463.098,A 0.000,B 0.000,C 90.000,E1 197.583} C_DIS
LIN {X 0.036,Y -138.352,Z 463.056,A 0.000,B 0.000,C 90.000,E1 190.074} C_DIS
LIN {X 0.009,Y -139.531,Z 463.004,A 0.000,B 0.000,C 90.000,E1 180.745} C_DIS
LIN {X -0.038,Y -141.212,Z 462.973,A 0.000,B 0.000,C 90.000,E1 175.179} C_DIS
LIN {X 0.062,Y -142.586,Z 462.958,A 0.000,B 0.000,C 90.000,E1 172.356} C_DIS
LIN {X 0.016,Y -144.884,Z 462.932,A 0.000,B 0.000,C 90.000,E1 167.757} C_DIS
LIN {X -0.030,Y -147.510,Z 462.912,A 0.000,B 0.000,C 90.000,E1 164.102} C_DIS
LIN {X 0.045,Y -150.104,Z 462.891,A 0.000,B 0.000,C 90.000,E1 160.423} C_DIS
LIN {X 0.056,Y -153.461,Z 462.871,A 0.000,B 0.000,C 90.000,E1 156.794} C_DIS
LIN {X -0.091,Y -157.825,Z 462.846,A 0.000,B 0.000,C 90.000,E1 152.359} C_DIS
LIN {X -0.061,Y -162.108,Z 462.827,A 0.000,B 0.000,C 90.000,E1 148.791} C_DIS
LIN {X -0.036,Y -166.309,Z 462.807,A 0.000,B 0.000,C 90.000,E1 145.261} C_DIS
LIN {X 0.066,Y -171.326,Z 462.788,A 0.000,B 0.000,C 90.000,E1 141.743} C_DIS
LIN {X -0.006,Y -176.226,Z 462.768,A 0.000,B 0.000,C 90.000,E1 138.324} C_DIS
LIN {X 0.114,Y -180.506,Z 462.754,A 0.000,B 0.000,C 90.000,E1 135.729} C_DIS
LIN {X 0.094,Y -185.909,Z 462.736,A 0.000,B 0.000,C 90.000,E1 132.366} C_DIS
LIN {X 0.030,Y -190.537,Z 462.722,A 0.000,B 0.000,C 90.000,E1 129.886} C_DIS
LIN {X -0.046,Y -194.389,Z 462.709,A 0.000,B 0.000,C 90.000,E1 127.649} C_DIS
LIN {X -0.109,Y -291.597,Z 462.709,A 0.000,B 0.000,C 90.000,E1 127.649} C_DIS
LIN {X 0.082,Y -292.602,Z 462.709,A 0.000,B 0.000,C 90.000,E1 127.604} C_DIS
LIN {X -0.114,Y -297.798,Z 462.708,A 0.000,B 0.000,C 90.000,E1 127.443} C_DIS
LIN {X 0.126,Y -300.732,Z 462.707,A 0.000,B 0.000,C 90.000,E1 127.156} C_DIS
LIN {X -0.058,Y -304.485,Z 462.704,A 0.000,B 0.000,C 90.000,E1 126.710} C_DIS
LIN {X -0.047,Y -306.288,Z 462.702,A 0.000,B 0.000,C 90.000,E1 126.377} C_DIS
LIN {X 0.146,Y -307.703,Z 462.700,A 0.000,B 0.000,C 90.000,E1 126.011} C_DIS
LIN {X -0.036,Y -311.769,Z 462.693,A 0.000,B 0.000,C 90.000,E1 124.739} C_DIS
LIN {X -0.026,Y -322.619,Z 462.675,A 0.000,B 0.000,C 90.000,E1 121.514} C_DIS
LIN {X -0.172,Y -333.765,Z 462.659,A 0.000,B 0.000,C 90.000,E1 118.693} C_DIS
LIN {X 0.149,Y -346.331,Z 462.644,A 0.000,B 0.000,C 90.000,E1 115.848} C_DIS
LIN {X -0.126,Y -358.780,Z 462.630,A 0.000,B 0.000,C 90.000,E1 113.462} C_DIS
LIN {X 0.105,Y -372.529,Z 462.617,A 0.000,B 0.000,C 90.000,E1 111.046} C_DIS
LIN {X 0.068,Y -387.676,Z 462.604,A 0.000,B 0.000,C 90.000,E1 108.725} C_DIS
LIN {X 0.161,Y -404.334,Z 462.591,A 0.000,B 0.000,C 90.000,E1 106.441} C_DIS
LIN {X 0.051,Y -422.625,Z 462.579,A 0.000,B 0.000,C 90.000,E1 104.245} C_DIS
LIN {X 0.057,Y -442.427,Z 462.567,A 0.000,B 0.000,C 90.000,E1 102.119} C_DIS
LIN {X -0.202,Y -462.874,Z 462.557,A 0.000,B 0.000,C 90.000,E1 100.197} C_DIS
LIN {X -0.150,Y -483.625,Z 462.547,A 0.000,B 0.000,C 90.000,E1 98.398} C_DIS
LIN {X -0.080,Y -485.565,Z 462.545,A 0.000,B 0.000,C 90.000,E1 98.163} C_DIS
LIN {X -0.077,Y -487.049,Z 462.544,A 0.000,B 0.000,C 90.000,E1 97.936} C_DIS
LIN {X -0.188,Y -488.283,Z 462.543,A 0.000,B 0.000,C 90.000,E1 97.701} C_DIS
LIN {X 0.184,Y -489.186,Z 462.541,A 0.000,B 0.000,C 90.000,E1 97.409} C_DIS
LIN {X -0.091,Y -490.153,Z 462.539,A 0.000,B 0.000,C 90.000,E1 96.947} C_DIS
LIN {X 0.127,Y -490.123,Z 462.536,A 0.000,B 0.000,C 90.000,E1 96.429} C_DIS
LIN {X -0.138,Y -489.089,Z 462.533,A 0.000,B 0.000,C 90.000,E1 95.967} C_DIS
LIN {X 0.192,Y -488.147,Z 462.532,A 0.000,B 0.000,C 90.000,E1 95.682} C_DIS
LIN {X 0.037,Y -486.865,Z 462.530,A 0.000,B 0.000,C 90.000,E1 95.454} C_DIS
LIN {X -0.235,Y -483.195,Z 462.528,A 0.000,B 0.000,C 90.000,E1 94.992} C_DIS
LIN {X -0.014,Y -459.509,Z 462.511,A 0.000,B 0.000,C 90.000,E1 91.949} C_DIS
LIN {X 0.213,Y -447.012,Z 462.501,A 0.000,B 0.000,C 90.000,E1 90.115} C_DIS
LIN {X 0.079,Y -432.070,Z 462.488,A 0.000,B 0.000,C 90.000,E1 87.764} C_DIS
LIN {X 0.001,Y -417.530,Z 462.474,A 0.000,B 0.000,C 90.000,E1 85.355} C_DIS
LIN {X 0.068,Y -403.457,Z 462.460,A 0.000,B 0.000,C 90.000,E1 82.875} C_DIS
LIN {X 0.140,Y -392.593,Z 462.450,A 0.000,B 0.000,C 90.000,E1 80.905} C_DIS
LIN {X 0.056,Y -381.816,Z 462.439,A 0.000,B 0.000,C 90.000,E1 78.926} C_DIS
LIN {X -0.106,Y -366.724,Z 462.422,A 0.000,B 0.000,C 90.000,E1 76.047} C_DIS
LIN {X -0.125,Y -356.827,Z 462.411,A 0.000,B 0.000,C 90.000,E1 73.976} C_DIS
LIN {X 0.137,Y -344.061,Z 462.394,A 0.000,B 0.000,C 90.000,E1 70.913} C_DIS
LIN {X 0.030,Y -332.474,Z 462.377,A 0.000,B 0.000,C 90.000,E1 67.847} C_DIS
LIN {X -0.081,Y -323.451,Z 462.363,A 0.000,B 0.000,C 90.000,E1 65.357} C_DIS
LIN {X -0.004,Y -314.656,Z 462.349,A 0.000,B 0.000,C 90.000,E1 62.794} C_DIS
LIN {X -0.032,Y -307.100,Z 462.336,A 0.000,B 0.000,C 90.000,E1 60.539} C_DIS
LIN {X 0.034,Y -296.640,Z 462.318,A 0.000,B 0.000,C 90.000,E1 57.248} C_DIS
LIN {X 0.018,Y -286.866,Z 462.300,A 0.000,B 0.000,C 90.000,E1 53.909} C_DIS
LIN {X -0.119,Y -281.258,Z 462.288,A 0.000,B 0.000,C 90.000,E1 51.904} C_DIS
LIN {X -0.014,Y -275.443,Z 462.277,A 0.000,B 0.000,C 90.000,E1 49.828} C_DIS
LIN {X -0.046,Y -269.344,Z 462.265,A 0.000,B 0.000,C 90.000,E1 47.757} C_DIS
LIN {X -0.011,Y -263.075,Z 462.254,A 0.000,B 0.000,C 90.000,E1 45.648} C_DIS
LIN {X -0.102,Y -256.629,Z 462.242,A 0.000,B 0.000,C 90.000,E1 43.542} C_DIS
LIN {X 0.052,Y -250.108,Z 462.230,A 0.000,B 0.000,C 90.000,E1 41.353} C_DIS
LIN {X -0.068,Y -239.406,Z 462.210,A 0.000,B 0.000,C 90.000,E1 37.729} C_DIS
LIN {X -0.016,Y -231.520,Z 462.193,A 0.000,B 0.000,C 90.000,E1 34.739} C_DIS
LIN {X -0.044,Y -224.333,Z 462.176,A 0.000,B 0.000,C 90.000,E1 31.720} C_DIS
LIN {X 0.087,Y -217.962,Z 462.159,A 0.000,B 0.000,C 90.000,E1 28.615} C_DIS
LIN {X -0.105,Y -211.243,Z 462.137,A 0.000,B 0.000,C 90.000,E1 24.771} C_DIS
LIN {X 0.006,Y -205.505,Z 462.116,A 0.000,B 0.000,C 90.000,E1 20.791} C_DIS
LIN {X -0.030,Y -200.795,Z 462.093,A 0.000,B 0.000,C 90.000,E1 16.804} C_DIS
LIN {X -0.047,Y -197.071,Z 462.071,A 0.000,B 0.000,C 90.000,E1 12.771} C_DIS
LIN {X -0.048,Y -193.465,Z 462.039,A 0.000,B 0.000,C 90.000,E1 7.068} C_DIS
LIN {X 0.070,Y -192.866,Z 461.961,A 0.000,B 0.000,C 90.000,E1 352.932} C_DIS
LIN {X -0.029,Y -196.201,Z 461.929,A 0.000,B 0.000,C 90.000,E1 347.229} C_DIS
LIN {X 0.046,Y -199.678,Z 461.906,A 0.000,B 0.000,C 90.000,E1 343.142} C_DIS
LIN {X -0.048,Y -204.045,Z 461.884,A 0.000,B 0.000,C 90.000,E1 339.135} C_DIS
LIN {X 0.103,Y -209.407,Z 461.862,A 0.000,B 0.000,C 90.000,E1 335.101} C_DIS
LIN {X 0.017,Y -215.585,Z 461.840,A 0.000,B 0.000,C 90.000,E1 331.179} C_DIS
LIN {X -0.031,Y -220.975,Z 461.823,A 0.000,B 0.000,C 90.000,E1 328.074} C_DIS
LIN {X 0.087,Y -228.195,Z 461.801,A 0.000,B 0.000,C 90.000,E1 324.196} C_DIS
LIN {X -0.033,Y -236.121,Z 461.780,A 0.000,B 0.000,C 90.000,E1 320.436} C_DIS
LIN {X 0.002,Y -245.149,Z 461.759,A 0.000,B 0.000,C 90.000,E1 316.701} C_DIS
LIN {X -0.036,Y -254.393,Z 461.741,A 0.000,B 0.000,C 90.000,E1 313.419} C_DIS
LIN {X 0.051,Y -264.813,Z 461.723,A 0.000,B 0.000,C 90.000,E1 310.172} C_DIS
LIN {X -0.035,Y -276.255,Z 461.706,A 0.000,B 0.000,C 90.000,E1 307.030} C_DIS
LIN {X -0.034,Y -287.133,Z 461.690,A 0.000,B 0.000,C 90.000,E1 304.278} C_DIS
LIN {X -0.085,Y -300.161,Z 461.674,A 0.000,B 0.000,C 90.000,E1 301.258} C_DIS
LIN {X -0.074,Y -315.564,Z 461.655,A 0.000,B 0.000,C 90.000,E1 297.975} C_DIS
LIN {X -0.004,Y -327.498,Z 461.643,A 0.000,B 0.000,C 90.000,E1 295.720} C_DIS
LIN {X 0.039,Y -342.266,Z 461.629,A 0.000,B 0.000,C 90.000,E1 293.206} C_DIS
LIN {X -0.029,Y -362.965,Z 461.612,A 0.000,B 0.000,C 90.000,E1 290.174} C_DIS
LIN {X -0.121,Y -388.641,Z 461.594,A 0.000,B 0.000,C 90.000,E1 286.968} C_DIS
LIN {X 0.046,Y -408.620,Z 461.582,A 0.000,B 0.000,C 90.000,E1 284.717} C_DIS
LIN {X 0.021,Y -429.223,Z 461.570,A 0.000,B 0.000,C 90.000,E1 282.647} C_DIS
LIN {X 0.172,Y -439.177,Z 461.565,A 0.000,B 0.000,C 90.000,E1 281.602} C_DIS
LIN {X -0.009,Y -446.513,Z 461.560,A 0.000,B 0.000,C 90.000,E1 280.838} C_DIS
LIN {X -0.016,Y -455.608,Z 461.554,A 0.000,B 0.000,C 90.000,E1 279.792} C_DIS
LIN {X 0.086,Y -463.827,Z 461.549,A 0.000,B 0.000,C 90.000,E1 278.746} C_DIS
LIN {X -0.025,Y -469.341,Z 461.544,A 0.000,B 0.000,C 90.000,E1 277.992} C_DIS
LIN {X -0.085,Y -474.229,Z 461.540,A 0.000,B 0.000,C 90.000,E1 277.239} C_DIS
LIN {X -0.113,Y -478.624,Z 461.536,A 0.000,B 0.000,C 90.000,E1 276.486} C_DIS
LIN {X -0.151,Y -482.569,Z 461.532,A 0.000,B 0.000,C 90.000,E1 275.739} C_DIS
LIN {X -0.156,Y -485.911,Z 461.528,A 0.000,B 0.000,C 90.000,E1 274.992} C_DIS
LIN {X 0.035,Y -487.804,Z 461.525,A 0.000,B 0.000,C 90.000,E1 274.473} C_DIS
LIN {X 0.231,Y -489.311,Z 461.522,A 0.000,B 0.000,C 90.000,E1 273.955} C_DIS
LIN {X -0.084,Y -490.484,Z 461.519,A 0.000,B 0.000,C 90.000,E1 273.498} C_DIS
LIN {X 0.129,Y -491.248,Z 461.517,A 0.000,B 0.000,C 90.000,E1 272.980} C_DIS
LIN {X -0.168,Y -491.627,Z 461.514,A 0.000,B 0.000,C 90.000,E1 272.522} C_DIS
LIN {X 0.033,Y -491.598,Z 461.511,A 0.000,B 0.000,C 90.000,E1 272.007} C_DIS
LIN {X -0.239,Y -491.155,Z 461.508,A 0.000,B 0.000,C 90.000,E1 271.547} C_DIS
LIN {X -0.036,Y -490.237,Z 461.506,A 0.000,B 0.000,C 90.000,E1 271.031} C_DIS
LIN {X 0.166,Y -488.845,Z 461.503,A 0.000,B 0.000,C 90.000,E1 270.516} C_DIS
LIN {X -0.126,Y -486.931,Z 461.500,A 0.000,B 0.000,C 90.000,E1 270.057} C_DIS
LIN {X 0.062,Y -484.336,Z 461.497,A 0.000,B 0.000,C 90.000,E1 269.542} C_DIS
LIN {X 0.229,Y -481.017,Z 461.495,A 0.000,B 0.000,C 90.000,E1 269.026} C_DIS
LIN {X -0.101,Y -476.795,Z 461.492,A 0.000,B 0.000,C 90.000,E1 268.568} C_DIS
LIN {X 0.041,Y -471.462,Z 461.489,A 0.000,B 0.000,C 90.000,E1 268.051} C_DIS
LIN {X 0.023,Y -465.408,Z 461.487,A 0.000,B 0.000,C 90.000,E1 267.593} C_DIS
LIN {X -0.201,Y -462.389,Z 461.486,A 0.000,B 0.000,C 90.000,E1 267.421} C_DIS
LIN {X 0.091,Y -455.844,Z 461.484,A 0.000,B 0.000,C 90.000,E1 267.020} C_DIS
LIN {X -0.070,Y -449.048,Z 461.482,A 0.000,B 0.000,C 90.000,E1 266.731} C_DIS
LIN {X 0.074,Y -441.976,Z 461.480,A 0.000,B 0.000,C 90.000,E1 266.445} C_DIS
LIN {X 0.186,Y -434.065,Z 461.479,A 0.000,B 0.000,C 90.000,E1 266.216} C_DIS
LIN {X -0.117,Y -425.275,Z 461.478,A 0.000,B 0.000,C 90.000,E1 266.102} C_DIS
LIN {X -0.051,Y -415.008,Z 461.478,A 0.000,B 0.000,C 90.000,E1 265.988} C_DIS
LIN {X 0.087,Y -405.845,Z 461.477,A 0.000,B 0.000,C 90.000,E1 265.927} C_DIS
LIN {X 0.017,Y -180.918,Z 461.477,A 0.000,B 0.000,C 90.000,E1 265.927} C_DIS
LIN {X -0.069,Y -180.871,Z 461.472,A 0.000,B 0.000,C 90.000,E1 265.065} C_DIS
LIN {X -0.012,Y -178.987,Z 461.444,A 0.000,B 0.000,C 90.000,E1 259.982} C_DIS
LIN {X 0.000,Y -177.967,Z 461.435,A 0.000,B 0.000,C 90.000,E1 258.285} C_DIS
LIN {X 0.018,Y -175.610,Z 461.411,A 0.000,B 0.000,C 90.000,E1 254.031} C_DIS
LIN {X 0.030,Y -172.333,Z 461.388,A 0.000,B 0.000,C 90.000,E1 249.752} C_DIS
LIN {X 0.009,Y -171.809,Z 461.383,A 0.000,B 0.000,C 90.000,E1 248.901} C_DIS
LIN {X 0.017,Y -170.271,Z 461.373,A 0.000,B 0.000,C 90.000,E1 247.177} C_DIS
LIN {X -0.047,Y -166.812,Z 461.349,A 0.000,B 0.000,C 90.000,E1 242.871} C_DIS
LIN {X 0.010,Y -162.795,Z 461.325,A 0.000,B 0.000,C 90.000,E1 238.486} C_DIS
LIN {X 0.070,Y -161.483,Z 461.315,A 0.000,B 0.000,C 90.000,E1 236.707} C_DIS
LIN {X -0.014,Y -157.478,Z 461.291,A 0.000,B 0.000,C 90.000,E1 232.316} C_DIS
LIN {X 0.043,Y -155.494,Z 461.276,A 0.000,B 0.000,C 90.000,E1 229.622} C_DIS
LIN {X -0.025,Y -151.799,Z 461.251,A 0.000,B 0.000,C 90.000,E1 225.162} C_DIS
LIN {X -0.012,Y -150.009,Z 461.236,A 0.000,B 0.000,C 90.000,E1 222.447} C_DIS
LIN {X 0.020,Y -146.835,Z 461.211,A 0.000,B 0.000,C 90.000,E1 217.890} C_DIS
LIN {X 0.006,Y -145.417,Z 461.195,A 0.000,B 0.000,C 90.000,E1 215.152} C_DIS
LIN {X 0.041,Y -142.845,Z 461.170,A 0.000,B 0.000,C 90.000,E1 210.541} C_DIS
LIN {X -0.028,Y -141.459,Z 461.149,A 0.000,B 0.000,C 90.000,E1 206.873} C_DIS
LIN {X 0.011,Y -139.374,Z 461.113,A 0.000,B 0.000,C 90.000,E1 200.355} C_DIS
LIN {X -0.048,Y -138.825,Z 461.098,A 0.000,B 0.000,C 90.000,E1 197.583} C_DIS
LIN {X 0.041,Y -138.352,Z 461.056,A 0.000,B 0.000,C 90.000,E1 190.074} C_DIS
LIN {X 0.015,Y -139.531,Z 461.004,A 0.000,B 0.000,C 90.000,E1 180.745} C_DIS
LIN {X -0.033,Y -141.210,Z 460.973,A 0.000,B 0.000,C 90.000,E1 175.179} C_DIS
LIN {X 0.068,Y -142.585,Z 460.958,A 0.000,B 0.000,C 90.000,E1 172.356} C_DIS
LIN {X 0.022,Y -144.882,Z 460.932,A 0.000,B 0.000,C 90.000,E1 167.757} C_DIS
LIN {X -0.025,Y -147.509,Z 460.912,A 0.000,B 0.000,C 90.000,E1 164.102} C_DIS
LIN {X 0.050,Y -150.102,Z 460.891,A 0.000,B 0.000,C 90.000,E1 160.423} C_DIS
LIN {X 0.062,Y -153.459,Z 460.871,A 0.000,B 0.000,C 90.000,E1 156.794} C_DIS
LIN {X -0.086,Y -157.822,Z 460.846,A 0.000,B 0.000,C 90.000,E1 152.359} C_DIS
LIN {X -0.054,Y -162.105,Z 460.827,A 0.000,B 0.000,C 90.000,E1 148.791} C_DIS
LIN {X -0.030,Y -166.307,Z 460.807,A 0.000,B 0.000,C 90.000,E1 145.261} C_DIS
LIN {X -0.034,Y -171.323,Z 460.788,A 0.000,B 0.000,C 90.000,E1 141.778} C_DIS
LIN {X 0.000,Y -176.224,Z 460.768,A 0.000,B 0.000,C 90.000,E1 138.324} C_DIS
LIN {X -0.006,Y -180.502,Z 460.754,A 0.000,B 0.000,C 90.000,E1 135.769} C_DIS
LIN {X -0.024,Y -185.906,Z 460.736,A 0.000,B 0.000,C 90.000,E1 132.405} C_DIS
LIN {X 0.036,Y -190.533,Z 460.722,A 0.000,B 0.000,C 90.000,E1 129.886} C_DIS
LIN {X 0.031,Y -194.491,Z 460.709,A 0.000,B 0.000,C 90.000,E1 127.569} C_DIS
LIN {X 0.012,Y -291.941,Z 460.709,A 0.000,B 0.000,C 90.000,E1 127.569} C_DIS
LIN {X -0.104,Y -296.970,Z 460.708,A 0.000,B 0.000,C 90.000,E1 127.443} C_DIS
LIN {X -0.128,Y -299.937,Z 460.707,A 0.000,B 0.000,C 90.000,E1 127.237} C_DIS
LIN {X -0.019,Y -303.680,Z 460.704,A 0.000,B 0.000,C 90.000,E1 126.790} C_DIS
LIN {X 0.087,Y -305.601,Z 460.703,A 0.000,B 0.000,C 90.000,E1 126.457} C_DIS
LIN {X -0.051,Y -307.115,Z 460.701,A 0.000,B 0.000,C 90.000,E1 126.171} C_DIS
LIN {X 0.159,Y -308.380,Z 460.699,A 0.000,B 0.000,C 90.000,E1 125.804} C_DIS
LIN {X 0.048,Y -319.879,Z 460.679,A 0.000,B 0.000,C 90.000,E1 122.260} C_DIS
LIN {X -0.010,Y -330.668,Z 460.663,A 0.000,B 0.000,C 90.000,E1 119.411} C_DIS
LIN {X -0.079,Y -342.849,Z 460.648,A 0.000,B 0.000,C 90.000,E1 116.616} C_DIS
LIN {X 0.021,Y -354.931,Z 460.634,A 0.000,B 0.000,C 90.000,E1 114.155} C_DIS
LIN {X -0.043,Y -368.283,Z 460.621,A 0.000,B 0.000,C 90.000,E1 111.770} C_DIS
LIN {X 0.162,Y -383.004,Z 460.608,A 0.000,B 0.000,C 90.000,E1 109.396} C_DIS
LIN {X -0.119,Y -399.201,Z 460.595,A 0.000,B 0.000,C 90.000,E1 107.149} C_DIS
LIN {X 0.026,Y -416.993,Z 460.583,A 0.000,B 0.000,C 90.000,E1 104.898} C_DIS
LIN {X -0.245,Y -436.443,Z 460.571,A 0.000,B 0.000,C 90.000,E1 102.771} C_DIS
LIN {X 0.153,Y -456.726,Z 460.560,A 0.000,B 0.000,C 90.000,E1 100.715} C_DIS
LIN {X -0.029,Y -480.158,Z 460.548,A 0.000,B 0.000,C 90.000,E1 98.681} C_DIS
LIN {X 0.046,Y -482.785,Z 460.547,A 0.000,B 0.000,C 90.000,E1 98.454} C_DIS
LIN {X 0.193,Y -484.902,Z 460.546,A 0.000,B 0.000,C 90.000,E1 98.219} C_DIS
LIN {X -0.210,Y -486.522,Z 460.545,A 0.000,B 0.000,C 90.000,E1 98.049} C_DIS
LIN {X 0.160,Y -487.934,Z 460.543,A 0.000,B 0.000,C 90.000,E1 97.757} C_DIS
LIN {X -0.017,Y -488.984,Z 460.542,A 0.000,B 0.000,C 90.000,E1 97.530} C_DIS
LIN {X 0.196,Y -490.198,Z 460.539,A 0.000,B 0.000,C 90.000,E1 97.011} C_DIS
LIN {X -0.072,Y -490.392,Z 460.536,A 0.000,B 0.000,C 90.000,E1 96.549} C_DIS
LIN {X 0.154,Y -489.597,Z 460.534,A 0.000,B 0.000,C 90.000,E1 96.030} C_DIS
LIN {X -0.106,Y -487.677,Z 460.531,A 0.000,B 0.000,C 90.000,E1 95.568} C_DIS
LIN {X -0.215,Y -486.175,Z 460.529,A 0.000,B 0.000,C 90.000,E1 95.334} C_DIS
LIN {X 0.136,Y -478.247,Z 460.524,A 0.000,B 0.000,C 90.000,E1 94.302} C_DIS
LIN {X 0.151,Y -458.649,Z 460.510,A 0.000,B 0.000,C 90.000,E1 91.776} C_DIS
LIN {X -0.098,Y -446.235,Z 460.500,A 0.000,B 0.000,C 90.000,E1 90.000} C_DIS
LIN {X 0.184,Y -431.322,Z 460.487,A 0.000,B 0.000,C 90.000,E1 87.593} C_DIS
LIN {X 0.120,Y -416.797,Z 460.473,A 0.000,B 0.000,C 90.000,E1 85.179} C_DIS
LIN {X 0.119,Y -402.747,Z 460.460,A 0.000,B 0.000,C 90.000,E1 82.704} C_DIS
LIN {X 0.107,Y -393.451,Z 460.450,A 0.000,B 0.000,C 90.000,E1 81.027} C_DIS
LIN {X 0.032,Y -382.678,Z 460.439,A 0.000,B 0.000,C 90.000,E1 79.050} C_DIS
LIN {X -0.114,Y -367.585,Z 460.423,A 0.000,B 0.000,C 90.000,E1 76.172} C_DIS
LIN {X -0.066,Y -356.296,Z 460.410,A 0.000,B 0.000,C 90.000,E1 73.795} C_DIS
LIN {X 0.178,Y -343.579,Z 460.393,A 0.000,B 0.000,C 90.000,E1 70.732} C_DIS
LIN {X 0.053,Y -331.968,Z 460.376,A 0.000,B 0.000,C 90.000,E1 67.667} C_DIS
LIN {X 0.010,Y -321.817,Z 460.360,A 0.000,B 0.000,C 90.000,E1 64.845} C_DIS
LIN {X -0.016,Y -314.098,Z 460.348,A 0.000,B 0.000,C 90.000,E1 62.615} C_DIS
LIN {X 0.135,Y -305.427,Z 460.333,A 0.000,B 0.000,C 90.000,E1 59.999} C_DIS
LIN {X 0.121,Y -297.062,Z 460.319,A 0.000,B 0.000,C 90.000,E1 57.375} C_DIS
LIN {X -0.048,Y -287.241,Z 460.300,A 0.000,B 0.000,C 90.000,E1 54.069} C_DIS
LIN {X -0.009,Y -281.600,Z 460.289,A 0.000,B 0.000,C 90.000,E1 52.029} C_DIS
LIN {X -0.071,Y -275.808,Z 460.278,A 0.000,B 0.000,C 90.000,E1 49.989} C_DIS
LIN {X -0.096,Y -269.737,Z 460.266,A 0.000,B 0.000,C 90.000,E1 47.919} C_DIS
LIN {X -0.055,Y -263.494,Z 460.254,A 0.000,B 0.000,C 90.000,E1 45.810} C_DIS
LIN {X -0.137,Y -257.089,Z 460.243,A 0.000,B 0.000,C 90.000,E1 43.704} C_DIS
LIN {X 0.029,Y -250.576,Z 460.231,A 0.000,B 0.000,C 90.000,E1 41.515} C_DIS
LIN {X -0.065,Y -241.943,Z 460.214,A 0.000,B 0.000,C 90.000,E1 38.624} C_DIS
LIN {X 0.006,Y -233.862,Z 460.198,A 0.000,B 0.000,C 90.000,E1 35.644} C_DIS
LIN {X 0.035,Y -226.462,Z 460.181,A 0.000,B 0.000,C 90.000,E1 32.625} C_DIS
LIN {X -0.046,Y -219.786,Z 460.164,A 0.000,B 0.000,C 90.000,E1 29.589} C_DIS
LIN {X -0.044,Y -214.095,Z 460.147,A 0.000,B 0.000,C 90.000,E1 26.488} C_DIS
LIN {X 0.130,Y -207.906,Z 460.125,A 0.000,B 0.000,C 90.000,E1 22.514} C_DIS
LIN {X 0.101,Y -202.736,Z 460.103,A 0.000,B 0.000,C 90.000,E1 18.544} C_DIS
LIN {X 0.050,Y -198.557,Z 460.081,A 0.000,B 0.000,C 90.000,E1 14.537} C_DIS
LIN {X 0.035,Y -194.862,Z 460.054,A 0.000,B 0.000,C 90.000,E1 9.670} C_DIS
LIN {X -0.012,Y -192.187,Z 460.022,A 0.000,B 0.000,C 90.000,E1 3.955} C_DIS
LIN {X 0.002,Y -193.111,Z 459.956,A 0.000,B 0.000,C 90.000,E1 352.129} C_DIS
LIN {X -0.023,Y -196.660,Z 459.924,A 0.000,B 0.000,C 90.000,E1 346.408} C_DIS
LIN {X -0.076,Y -200.310,Z 459.902,A 0.000,B 0.000,C 90.000,E1 342.362} C_DIS
LIN {X 0.107,Y -204.864,Z 459.880,A 0.000,B 0.000,C 90.000,E1 338.284} C_DIS
LIN {X -0.015,Y -210.424,Z 459.857,A 0.000,B 0.000,C 90.000,E1 334.332} C_DIS
LIN {X 0.033,Y -216.775,Z 459.836,A 0.000,B 0.000,C 90.000,E1 330.383} C_DIS
LIN {X 0.033,Y -223.632,Z 459.814,A 0.000,B 0.000,C 90.000,E1 326.501} C_DIS
LIN {X 0.109,Y -229.566,Z 459.797,A 0.000,B 0.000,C 90.000,E1 323.417} C_DIS
LIN {X -0.003,Y -237.729,Z 459.776,A 0.000,B 0.000,C 90.000,E1 319.666} C_DIS
LIN {X -0.091,Y -246.962,Z 459.755,A 0.000,B 0.000,C 90.000,E1 315.972} C_DIS
LIN {X -0.072,Y -256.495,Z 459.737,A 0.000,B 0.000,C 90.000,E1 312.690} C_DIS
LIN {X -0.039,Y -268.397,Z 459.717,A 0.000,B 0.000,C 90.000,E1 309.116} C_DIS
LIN {X 0.022,Y -280.267,Z 459.700,A 0.000,B 0.000,C 90.000,E1 305.964} C_DIS
LIN {X 0.093,Y -294.249,Z 459.681,A 0.000,B 0.000,C 90.000,E1 302.546} C_DIS
LIN {X -0.101,Y -306.145,Z 459.666,A 0.000,B 0.000,C 90.000,E1 299.922} C_DIS
LIN {X -0.043,Y -318.877,Z 459.652,A 0.000,B 0.000,C 90.000,E1 297.308} C_DIS
LIN {X -0.012,Y -336.600,Z 459.634,A 0.000,B 0.000,C 90.000,E1 294.131} C_DIS
LIN {X -0.045,Y -348.307,Z 459.624,A 0.000,B 0.000,C 90.000,E1 292.280} C_DIS
LIN {X -0.069,Y -365.227,Z 459.610,A 0.000,B 0.000,C 90.000,E1 289.866} C_DIS
LIN {X 0.146,Y -388.681,Z 459.594,A 0.000,B 0.000,C 90.000,E1 286.913} C_DIS
LIN {X -0.102,Y -405.995,Z 459.583,A 0.000,B 0.000,C 90.000,E1 285.009} C_DIS
LIN {X 0.053,Y -426.820,Z 459.572,A 0.000,B 0.000,C 90.000,E1 282.883} C_DIS
LIN {X -0.055,Y -436.808,Z 459.566,A 0.000,B 0.000,C 90.000,E1 281.883} C_DIS
LIN {X 0.099,Y -446.411,Z 459.560,A 0.000,B 0.000,C 90.000,E1 280.838} C_DIS
LIN {X 0.092,Y -455.518,Z 459.554,A 0.000,B 0.000,C 90.000,E1 279.792} C_DIS
LIN {X 0.196,Y -463.778,Z 459.549,A 0.000,B 0.000,C 90.000,E1 278.746} C_DIS
LIN {X 0.085,Y -469.273,Z 459.544,A 0.000,B 0.000,C 90.000,E1 277.992} C_DIS
LIN {X 0.025,Y -474.201,Z 459.540,A 0.000,B 0.000,C 90.000,E1 277.239} C_DIS
LIN {X -0.001,Y -478.613,Z 459.536,A 0.000,B 0.000,C 90.000,E1 276.486} C_DIS
LIN {X -0.039,Y -482.593,Z 459.532,A 0.000,B 0.000,C 90.000,E1 275.739} C_DIS
LIN {X -0.043,Y -485.999,Z 459.528,A 0.000,B 0.000,C 90.000,E1 274.992} C_DIS
LIN {X 0.149,Y -487.901,Z 459.525,A 0.000,B 0.000,C 90.000,E1 274.473} C_DIS
LIN {X -0.142,Y -489.423,Z 459.522,A 0.000,B 0.000,C 90.000,E1 274.012} C_DIS
LIN {X 0.032,Y -490.575,Z 459.519,A 0.000,B 0.000,C 90.000,E1 273.498} C_DIS
LIN {X 0.245,Y -491.346,Z 459.517,A 0.000,B 0.000,C 90.000,E1 272.980} C_DIS
LIN {X -0.051,Y -491.716,Z 459.514,A 0.000,B 0.000,C 90.000,E1 272.522} C_DIS
LIN {X 0.151,Y -491.675,Z 459.511,A 0.000,B 0.000,C 90.000,E1 272.007} C_DIS
LIN {X -0.121,Y -491.259,Z 459.509,A 0.000,B 0.000,C 90.000,E1 271.547} C_DIS
LIN {X 0.083,Y -490.373,Z 459.506,A 0.000,B 0.000,C 90.000,E1 271.031} C_DIS
LIN {X -0.205,Y -489.000,Z 459.503,A 0.000,B 0.000,C 90.000,E1 270.573} C_DIS
LIN {X -0.007,Y -487.094,Z 459.500,A 0.000,B 0.000,C 90.000,E1 270.057} C_DIS
LIN {X 0.181,Y -484.559,Z 459.498,A 0.000,B 0.000,C 90.000,E1 269.542} C_DIS
LIN {X -0.132,Y -481.243,Z 459.495,A 0.000,B 0.000,C 90.000,E1 269.083} C_DIS
LIN {X 0.019,Y -477.025,Z 459.492,A 0.000,B 0.000,C 90.000,E1 268.568} C_DIS
LIN {X -0.155,Y -474.573,Z 459.491,A 0.000,B 0.000,C 90.000,E1 268.339} C_DIS
LIN {X 0.157,Y -468.945,Z 459.488,A 0.000,B 0.000,C 90.000,E1 267.822} C_DIS
LIN {X -0.058,Y -462.764,Z 459.486,A 0.000,B 0.000,C 90.000,E1 267.421} C_DIS
LIN {X 0.196,Y -456.213,Z 459.484,A 0.000,B 0.000,C 90.000,E1 267.020} C_DIS
LIN {X -0.015,Y -449.408,Z 459.482,A 0.000,B 0.000,C 90.000,E1 266.731} C_DIS
LIN {X 0.141,Y -442.317,Z 459.480,A 0.000,B 0.000,C 90.000,E1 266.445} C_DIS
LIN {X -0.181,Y -434.528,Z 459.479,A 0.000,B 0.000,C 90.000,E1 266.274} C_DIS
LIN {X -0.086,Y -425.759,Z 459.478,A 0.000,B 0.000,C 90.000,E1 266.102} C_DIS
LIN {X -0.045,Y -415.180,Z 459.478,A 0.000,B 0.000,C 90.000,E1 265.988} C_DIS
LIN {X 0.089,Y -405.027,Z 459.477,A 0.000,B 0.000,C 90.000,E1 265.927} C_DIS
LIN {X 0.020,Y -180.918,Z 459.477,A 0.000,B 0.000,C 90.000,E1 265.927} C_DIS
LIN {X -0.061,Y -180.872,Z 459.472,A 0.000,B 0.000,C 90.000,E1 265.065} C_DIS
LIN {X -0.004,Y -178.988,Z 459.444,A 0.000,B 0.000,C 90.000,E1 259.982} C_DIS
LIN {X 0.007,Y -177.968,Z 459.435,A 0.000,B 0.000,C 90.000,E1 258.285} C_DIS
LIN {X 0.026,Y -175.612,Z 459.411,A 0.000,B 0.000,C 90.000,E1 254.031} C_DIS
LIN {X 0.038,Y -172.334,Z 459.388,A 0.000,B 0.000,C 90.000,E1 249.752} C_DIS
LIN {X 0.017,Y -171.810,Z 459.383,A 0.000,B 0.000,C 90.000,E1 248.901} C_DIS
LIN {X 0.024,Y -170.273,Z 459.373,A 0.000,B 0.000,C 90.000,E1 247.177} C_DIS
LIN {X -0.040,Y -166.815,Z 459.349,A 0.000,B 0.000,C 90.000,E1 242.871} C_DIS
LIN {X 0.018,Y -162.797,Z 459.325,A 0.000,B 0.000,C 90.000,E1 238.486} C_DIS
LIN {X 0.078,Y -161.483,Z 459.315,A 0.000,B 0.000,C 90.000,E1 236.707} C_DIS
LIN {X -0.007,Y -157.480,Z 459.291,A 0.000,B 0.000,C 90.000,E1 232.316} C_DIS
LIN {X 0.050,Y -155.496,Z 459.276,A 0.000,B 0.000,C 90.000,E1 229.622} C_DIS
LIN {X -0.017,Y -151.802,Z 459.251,A 0.000,B 0.000,C 90.000,E1 225.162} C_DIS
LIN {X -0.005,Y -150.012,Z 459.236,A 0.000,B 0.000,C 90.000,E1 222.447} C_DIS
LIN {X 0.026,Y -146.837,Z 459.211,A 0.000,B 0.000,C 90.000,E1 217.890} C_DIS
LIN {X 0.013,Y -145.418,Z 459.195,A 0.000,B 0.000,C 90.000,E1 215.152} C_DIS
LIN {X 0.048,Y -142.846,Z 459.170,A 0.000,B 0.000,C 90.000,E1 210.541} C_DIS
LIN {X -0.022,Y -141.460,Z 459.149,A 0.000,B 0.000,C 90.000,E1 206.873} C_DIS
LIN {X 0.017,Y -139.375,Z 459.113,A 0.000,B 0.000,C 90.000,E1 200.355} C_DIS
LIN {X -0.041,Y -138.826,Z 459.098,A 0.000,B 0.000,C 90.000,E1 197.583} C_DIS
LIN {X 0.048,Y -138.353,Z 459.056,A 0.000,B 0.000,C 90.000,E1 190.074} C_DIS
LIN {X 0.021,Y -139.530,Z 459.004,A 0.000,B 0.000,C 90.000,E1 180.745} C_DIS
LIN {X -0.026,Y -141.210,Z 458.973,A 0.000,B 0.000,C 90.000,E1 175.179} C_DIS
LIN {X -0.067,Y -142.584,Z 458.958,A 0.000,B 0.000,C 90.000,E1 172.413} C_DIS
LIN {X 0.028,Y -144.880,Z 458.932,A 0.000,B 0.000,C 90.000,E1 167.757} C_DIS
LIN {X -0.018,Y -147.508,Z 458.912,A 0.000,B 0.000,C 90.000,E1 164.102} C_DIS
LIN {X 0.057,Y -150.100,Z 458.891,A 0.000,B 0.000,C 90.000,E1 160.423} C_DIS
LIN {X 0.070,Y -153.456,Z 458.871,A 0.000,B 0.000,C 90.000,E1 156.794} C_DIS
LIN {X -0.079,Y -157.819,Z 458.846,A 0.000,B 0.000,C 90.000,E1 152.359} C_DIS
LIN {X -0.047,Y -162.102,Z 458.827,A 0.000,B 0.000,C 90.000,E1 148.791} C_DIS
LIN {X -0.022,Y -166.302,Z 458.807,A 0.000,B 0.000,C 90.000,E1 145.261} C_DIS
LIN {X -0.026,Y -171.320,Z 458.788,A 0.000,B 0.000,C 90.000,E1 141.778} C_DIS
LIN {X 0.008,Y -176.219,Z 458.768,A 0.000,B 0.000,C 90.000,E1 138.324} C_DIS
LIN {X 0.003,Y -180.498,Z 458.754,A 0.000,B 0.000,C 90.000,E1 135.769} C_DIS
LIN {X -0.016,Y -185.901,Z 458.736,A 0.000,B 0.000,C 90.000,E1 132.405} C_DIS
LIN {X 0.045,Y -190.528,Z 458.722,A 0.000,B 0.000,C 90.000,E1 129.886} C_DIS
LIN {X -0.030,Y -194.605,Z 458.708,A 0.000,B 0.000,C 90.000,E1 127.523} C_DIS
LIN {X -0.081,Y -292.644,Z 458.708,A 0.000,B 0.000,C 90.000,E1 127.523} C_DIS
LIN {X -0.092,Y -295.830,Z 458.708,A 0.000,B 0.000,C 90.000,E1 127.443} C_DIS
LIN {X 0.108,Y -298.782,Z 458.707,A 0.000,B 0.000,C 90.000,E1 127.237} C_DIS
LIN {X -0.036,Y -302.444,Z 458.705,A 0.000,B 0.000,C 90.000,E1 126.916} C_DIS
LIN {X -0.071,Y -306.023,Z 458.702,A 0.000,B 0.000,C 90.000,E1 126.377} C_DIS
LIN {X 0.128,Y -307.555,Z 458.700,A 0.000,B 0.000,C 90.000,E1 126.011} C_DIS
LIN {X -0.103,Y -308.767,Z 458.698,A 0.000,B 0.000,C 90.000,E1 125.724} C_DIS
LIN {X -0.016,Y -319.177,Z 458.680,A 0.000,B 0.000,C 90.000,E1 122.467} C_DIS
LIN {X -0.094,Y -329.876,Z 458.664,A 0.000,B 0.000,C 90.000,E1 119.617} C_DIS
LIN {X -0.031,Y -341.960,Z 458.649,A 0.000,B 0.000,C 90.000,E1 116.796} C_DIS
LIN {X 0.080,Y -355.531,Z 458.634,A 0.000,B 0.000,C 90.000,E1 114.027} C_DIS
LIN {X -0.106,Y -368.948,Z 458.620,A 0.000,B 0.000,C 90.000,E1 111.663} C_DIS
LIN {X -0.109,Y -383.738,Z 458.607,A 0.000,B 0.000,C 90.000,E1 109.322} C_DIS
LIN {X -0.129,Y -400.010,Z 458.595,A 0.000,B 0.000,C 90.000,E1 107.040} C_DIS
LIN {X 0.153,Y -417.883,Z 458.582,A 0.000,B 0.000,C 90.000,E1 104.773} C_DIS
LIN {X -0.068,Y -437.383,Z 458.570,A 0.000,B 0.000,C 90.000,E1 102.647} C_DIS
LIN {X -0.138,Y -457.693,Z 458.559,A 0.000,B 0.000,C 90.000,E1 100.658} C_DIS
LIN {X -0.181,Y -483.675,Z 458.547,A 0.000,B 0.000,C 90.000,E1 98.398} C_DIS
LIN {X -0.009,Y -485.595,Z 458.545,A 0.000,B 0.000,C 90.000,E1 98.163} C_DIS
LIN {X -0.192,Y -487.285,Z 458.544,A 0.000,B 0.000,C 90.000,E1 97.936} C_DIS
LIN {X 0.176,Y -488.552,Z 458.543,A 0.000,B 0.000,C 90.000,E1 97.644} C_DIS
LIN {X -0.101,Y -490.112,Z 458.540,A 0.000,B 0.000,C 90.000,E1 97.182} C_DIS
LIN {X 0.114,Y -490.608,Z 458.537,A 0.000,B 0.000,C 90.000,E1 96.663} C_DIS
LIN {X -0.149,Y -490.121,Z 458.534,A 0.000,B 0.000,C 90.000,E1 96.201} C_DIS
LIN {X 0.079,Y -488.571,Z 458.532,A 0.000,B 0.000,C 90.000,E1 95.682} C_DIS
LIN {X -0.076,Y -487.315,Z 458.530,A 0.000,B 0.000,C 90.000,E1 95.454} C_DIS
LIN {X -0.184,Y -485.639,Z 458.529,A 0.000,B 0.000,C 90.000,E1 95.220} C_DIS
LIN {X 0.019,Y -475.605,Z 458.522,A 0.000,B 0.000,C 90.000,E1 93.955} C_DIS
LIN {X -0.062,Y -456.243,Z 458.508,A 0.000,B 0.000,C 90.000,E1 91.432} C_DIS
LIN {X -0.158,Y -442.371,Z 458.496,A 0.000,B 0.000,C 90.000,E1 89.370} C_DIS
LIN {X -0.117,Y -429.167,Z 458.485,A 0.000,B 0.000,C 90.000,E1 87.249} C_DIS
LIN {X 0.181,Y -414.721,Z 458.471,A 0.000,B 0.000,C 90.000,E1 84.780} C_DIS
LIN {X 0.074,Y -402.280,Z 458.459,A 0.000,B 0.000,C 90.000,E1 82.591} C_DIS
LIN {X 0.113,Y -393.019,Z 458.450,A 0.000,B 0.000,C 90.000,E1 80.905} C_DIS
LIN {X 0.033,Y -382.231,Z 458.439,A 0.000,B 0.000,C 90.000,E1 78.926} C_DIS
LIN {X -0.192,Y -368.672,Z 458.424,A 0.000,B 0.000,C 90.000,E1 76.353} C_DIS
LIN {X -0.119,Y -357.311,Z 458.411,A 0.000,B 0.000,C 90.000,E1 73.976} C_DIS
LIN {X 0.172,Y -343.270,Z 458.392,A 0.000,B 0.000,C 90.000,E1 70.604} C_DIS
LIN {X 0.060,Y -332.785,Z 458.377,A 0.000,B 0.000,C 90.000,E1 67.847} C_DIS
LIN {X -0.045,Y -323.694,Z 458.363,A 0.000,B 0.000,C 90.000,E1 65.357} C_DIS
LIN {X -0.043,Y -313.711,Z 458.347,A 0.000,B 0.000,C 90.000,E1 62.487} C_DIS
LIN {X 0.039,Y -306.054,Z 458.335,A 0.000,B 0.000,C 90.000,E1 60.205} C_DIS
LIN {X 0.041,Y -297.637,Z 458.320,A 0.000,B 0.000,C 90.000,E1 57.582} C_DIS
LIN {X -0.108,Y -287.753,Z 458.301,A 0.000,B 0.000,C 90.000,E1 54.276} C_DIS
LIN {X 0.028,Y -280.204,Z 458.286,A 0.000,B 0.000,C 90.000,E1 51.537} C_DIS
LIN {X 0.110,Y -274.338,Z 458.275,A 0.000,B 0.000,C 90.000,E1 49.461} C_DIS
LIN {X 0.053,Y -268.201,Z 458.263,A 0.000,B 0.000,C 90.000,E1 47.391} C_DIS
LIN {X -0.127,Y -261.961,Z 458.252,A 0.000,B 0.000,C 90.000,E1 45.324} C_DIS
LIN {X -0.051,Y -255.521,Z 458.240,A 0.000,B 0.000,C 90.000,E1 43.176} C_DIS
LIN {X 0.085,Y -249.037,Z 458.228,A 0.000,B 0.000,C 90.000,E1 40.987} C_DIS
LIN {X -0.048,Y -240.469,Z 458.212,A 0.000,B 0.000,C 90.000,E1 38.096} C_DIS
LIN {X 0.033,Y -232.500,Z 458.195,A 0.000,B 0.000,C 90.000,E1 35.105} C_DIS
LIN {X 0.034,Y -225.201,Z 458.178,A 0.000,B 0.000,C 90.000,E1 32.084} C_DIS
LIN {X 0.003,Y -218.703,Z 458.161,A 0.000,B 0.000,C 90.000,E1 29.027} C_DIS
LIN {X -0.013,Y -213.163,Z 458.144,A 0.000,B 0.000,C 90.000,E1 25.924} C_DIS
LIN {X 0.052,Y -207.091,Z 458.122,A 0.000,B 0.000,C 90.000,E1 21.972} C_DIS
LIN {X 0.006,Y -202.052,Z 458.100,A 0.000,B 0.000,C 90.000,E1 18.000} C_DIS
LIN {X 0.076,Y -198.021,Z 458.078,A 0.000,B 0.000,C 90.000,E1 13.953} C_DIS
LIN {X 0.011,Y -194.445,Z 458.051,A 0.000,B 0.000,C 90.000,E1 9.095} C_DIS
LIN {X -0.062,Y -191.929,Z 458.019,A 0.000,B 0.000,C 90.000,E1 3.383} C_DIS
LIN {X -0.004,Y -192.990,Z 457.956,A 0.000,B 0.000,C 90.000,E1 352.129} C_DIS
LIN {X -0.035,Y -196.516,Z 457.924,A 0.000,B 0.000,C 90.000,E1 346.408} C_DIS
LIN {X -0.093,Y -200.143,Z 457.902,A 0.000,B 0.000,C 90.000,E1 342.362} C_DIS
LIN {X 0.084,Y -204.691,Z 457.879,A 0.000,B 0.000,C 90.000,E1 338.284} C_DIS
LIN {X -0.043,Y -210.258,Z 457.857,A 0.000,B 0.000,C 90.000,E1 334.332} C_DIS
LIN {X -0.001,Y -216.625,Z 457.835,A 0.000,B 0.000,C 90.000,E1 330.383} C_DIS
LIN {X -0.007,Y -223.466,Z 457.814,A 0.000,B 0.000,C 90.000,E1 326.501} C_DIS
LIN {X 0.063,Y -229.415,Z 457.797,A 0.000,B 0.000,C 90.000,E1 323.417} C_DIS
LIN {X -0.054,Y -237.587,Z 457.776,A 0.000,B 0.000,C 90.000,E1 319.666} C_DIS
LIN {X -0.149,Y -246.839,Z 457.755,A 0.000,B 0.000,C 90.000,E1 315.972} C_DIS
LIN {X -0.136,Y -256.380,Z 457.737,A 0.000,B 0.000,C 90.000,E1 312.690} C_DIS
LIN {X -0.109,Y -268.322,Z 457.717,A 0.000,B 0.000,C 90.000,E1 309.116} C_DIS
LIN {X -0.053,Y -280.213,Z 457.700,A 0.000,B 0.000,C 90.000,E1 305.964} C_DIS
LIN {X 0.013,Y -294.235,Z 457.681,A 0.000,B 0.000,C 90.000,E1 302.546} C_DIS
LIN {X 0.112,Y -307.659,Z 457.664,A 0.000,B 0.000,C 90.000,E1 299.539} C_DIS
LIN {X 0.077,Y -320.580,Z 457.650,A 0.000,B 0.000,C 90.000,E1 296.950} C_DIS
LIN {X -0.123,Y -338.504,Z 457.632,A 0.000,B 0.000,C 90.000,E1 293.823} C_DIS
LIN {X -0.101,Y -352.432,Z 457.620,A 0.000,B 0.000,C 90.000,E1 291.663} C_DIS
LIN {X 0.175,Y -365.277,Z 457.610,A 0.000,B 0.000,C 90.000,E1 289.812} C_DIS
LIN {X 0.021,Y -391.242,Z 457.592,A 0.000,B 0.000,C 90.000,E1 286.622} C_DIS
LIN {X -0.089,Y -408.708,Z 457.582,A 0.000,B 0.000,C 90.000,E1 284.717} C_DIS
LIN {X 0.222,Y -426.620,Z 457.572,A 0.000,B 0.000,C 90.000,E1 282.883} C_DIS
LIN {X 0.074,Y -436.558,Z 457.566,A 0.000,B 0.000,C 90.000,E1 281.895} C_DIS
LIN {X -0.143,Y -446.201,Z 457.560,A 0.000,B 0.000,C 90.000,E1 280.894} C_DIS
LIN {X 0.114,Y -453.117,Z 457.556,A 0.000,B 0.000,C 90.000,E1 280.074} C_DIS
LIN {X -0.087,Y -459.587,Z 457.552,A 0.000,B 0.000,C 90.000,E1 279.321} C_DIS
LIN {X 0.221,Y -465.539,Z 457.547,A 0.000,B 0.000,C 90.000,E1 278.511} C_DIS
LIN {X 0.129,Y -470.849,Z 457.543,A 0.000,B 0.000,C 90.000,E1 277.757} C_DIS
LIN {X 0.075,Y -475.626,Z 457.539,A 0.000,B 0.000,C 90.000,E1 277.004} C_DIS
LIN {X 0.011,Y -479.902,Z 457.535,A 0.000,B 0.000,C 90.000,E1 276.258} C_DIS
LIN {X -0.017,Y -483.734,Z 457.531,A 0.000,B 0.000,C 90.000,E1 275.511} C_DIS
LIN {X 0.162,Y -486.032,Z 457.528,A 0.000,B 0.000,C 90.000,E1 274.992} C_DIS
LIN {X -0.131,Y -487.932,Z 457.525,A 0.000,B 0.000,C 90.000,E1 274.531} C_DIS
LIN {X 0.065,Y -489.512,Z 457.522,A 0.000,B 0.000,C 90.000,E1 274.012} C_DIS
LIN {X 0.239,Y -490.643,Z 457.520,A 0.000,B 0.000,C 90.000,E1 273.498} C_DIS
LIN {X -0.037,Y -491.411,Z 457.517,A 0.000,B 0.000,C 90.000,E1 273.037} C_DIS
LIN {X 0.157,Y -491.811,Z 457.514,A 0.000,B 0.000,C 90.000,E1 272.522} C_DIS
LIN {X -0.133,Y -491.786,Z 457.511,A 0.000,B 0.000,C 90.000,E1 272.064} C_DIS
LIN {X 0.088,Y -491.358,Z 457.509,A 0.000,B 0.000,C 90.000,E1 271.547} C_DIS
LIN {X -0.198,Y -490.502,Z 457.506,A 0.000,B 0.000,C 90.000,E1 271.088} C_DIS
LIN {X 0.005,Y -489.162,Z 457.503,A 0.000,B 0.000,C 90.000,E1 270.573} C_DIS
LIN {X 0.203,Y -487.289,Z 457.500,A 0.000,B 0.000,C 90.000,E1 270.057} C_DIS
LIN {X -0.095,Y -484.798,Z 457.498,A 0.000,B 0.000,C 90.000,E1 269.599} C_DIS
LIN {X 0.077,Y -481.554,Z 457.495,A 0.000,B 0.000,C 90.000,E1 269.083} C_DIS
LIN {X 0.228,Y -477.414,Z 457.492,A 0.000,B 0.000,C 90.000,E1 268.568} C_DIS
LIN {X -0.103,Y -472.198,Z 457.489,A 0.000,B 0.000,C 90.000,E1 268.108} C_DIS
LIN {X -0.133,Y -469.352,Z 457.488,A 0.000,B 0.000,C 90.000,E1 267.879} C_DIS
LIN {X 0.077,Y -463.142,Z 457.486,A 0.000,B 0.000,C 90.000,E1 267.421} C_DIS
LIN {X -0.152,Y -456.612,Z 457.484,A 0.000,B 0.000,C 90.000,E1 267.078} C_DIS
LIN {X 0.066,Y -449.800,Z 457.482,A 0.000,B 0.000,C 90.000,E1 266.731} C_DIS
LIN {X 0.203,Y -442.657,Z 457.480,A 0.000,B 0.000,C 90.000,E1 266.445} C_DIS
LIN {X -0.134,Y -434.976,Z 457.479,A 0.000,B 0.000,C 90.000,E1 266.274} C_DIS
LIN {X -0.049,Y -426.286,Z 457.478,A 0.000,B 0.000,C 90.000,E1 266.102} C_DIS
LIN {X -0.013,Y -415.855,Z 457.478,A 0.000,B 0.000,C 90.000,E1 265.988} C_DIS
LIN {X 0.117,Y -407.452,Z 457.477,A 0.000,B 0.000,C 90.000,E1 265.927} C_DIS
LIN {X 0.030,Y -180.918,Z 457.477,A 0.000,B 0.000,C 90.000,E1 265.927} C_DIS
LIN {X -0.063,Y -180.872,Z 457.472,A 0.000,B 0.000,C 90.000,E1 265.065} C_DIS
LIN {X -0.006,Y -178.987,Z 457.444,A 0.000,B 0.000,C 90.000,E1 259.982} C_DIS
LIN {X 0.005,Y -177.969,Z 457.435,A 0.000,B 0.000,C 90.000,E1 258.285} C_DIS
LIN {X 0.024,Y -175.611,Z 457.411,A 0.000,B 0.000,C 90.000,E1 254.031} C_DIS
LIN {X 0.036,Y -172.334,Z 457.388,A 0.000,B 0.000,C 90.000,E1 249.752} C_DIS
LIN {X 0.015,Y -171.810,Z 457.383,A 0.000,B 0.000,C 90.000,E1 248.901} C_DIS
LIN {X 0.022,Y -170.273,Z 457.373,A 0.000,B 0.000,C 90.000,E1 247.177} C_DIS
LIN {X -0.042,Y -166.814,Z 457.349,A 0.000,B 0.000,C 90.000,E1 242.871} C_DIS
LIN {X 0.015,Y -162.796,Z 457.325,A 0.000,B 0.000,C 90.000,E1 238.486} C_DIS
LIN {X 0.076,Y -161.484,Z 457.315,A 0.000,B 0.000,C 90.000,E1 236.707} C_DIS
LIN {X -0.009,Y -157.479,Z 457.291,A 0.000,B 0.000,C 90.000,E1 232.316} C_DIS
LIN {X 0.048,Y -155.496,Z 457.276,A 0.000,B 0.000,C 90.000,E1 229.622} C_DIS
LIN {X -0.019,Y -151.801,Z 457.251,A 0.000,B 0.000,C 90.000,E1 225.162} C_DIS
LIN {X -0.007,Y -150.011,Z 457.236,A 0.000,B 0.000,C 90.000,E1 222.447} C_DIS
LIN {X 0.025,Y -146.837,Z 457.211,A 0.000,B 0.000,C 90.000,E1 217.890} C_DIS
LIN {X 0.011,Y -145.418,Z 457.195,A 0.000,B 0.000,C 90.000,E1 215.152} C_DIS
LIN {X 0.047,Y -142.845,Z 457.170,A 0.000,B 0.000,C 90.000,E1 210.541} C_DIS
LIN {X -0.024,Y -141.460,Z 457.149,A 0.000,B 0.000,C 90.000,E1 206.873} C_DIS
LIN {X 0.016,Y -139.375,Z 457.113,A 0.000,B 0.000,C 90.000,E1 200.355} C_DIS
LIN {X -0.042,Y -138.825,Z 457.098,A 0.000,B 0.000,C 90.000,E1 197.583} C_DIS
LIN {X 0.046,Y -138.353,Z 457.056,A 0.000,B 0.000,C 90.000,E1 190.074} C_DIS
LIN {X 0.020,Y -139.531,Z 457.004,A 0.000,B 0.000,C 90.000,E1 180.745} C_DIS
LIN {X -0.027,Y -141.210,Z 456.973,A 0.000,B 0.000,C 90.000,E1 175.179} C_DIS
LIN {X 0.073,Y -142.584,Z 456.958,A 0.000,B 0.000,C 90.000,E1 172.356} C_DIS
LIN {X 0.026,Y -144.880,Z 456.932,A 0.000,B 0.000,C 90.000,E1 167.757} C_DIS
LIN {X -0.019,Y -147.507,Z 456.912,A 0.000,B 0.000,C 90.000,E1 164.102} C_DIS
LIN {X 0.055,Y -150.100,Z 456.891,A 0.000,B 0.000,C 90.000,E1 160.423} C_DIS
LIN {X 0.068,Y -153.457,Z 456.871,A 0.000,B 0.000,C 90.000,E1 156.794} C_DIS
LIN {X -0.080,Y -157.820,Z 456.846,A 0.000,B 0.000,C 90.000,E1 152.359} C_DIS
LIN {X -0.048,Y -162.103,Z 456.827,A 0.000,B 0.000,C 90.000,E1 148.791} C_DIS
LIN {X -0.024,Y -166.304,Z 456.807,A 0.000,B 0.000,C 90.000,E1 145.261} C_DIS
LIN {X -0.028,Y -171.321,Z 456.788,A 0.000,B 0.000,C 90.000,E1 141.778} C_DIS
LIN {X 0.006,Y -176.220,Z 456.768,A 0.000,B 0.000,C 90.000,E1 138.324} C_DIS
LIN {X 0.001,Y -180.498,Z 456.754,A 0.000,B 0.000,C 90.000,E1 135.769} C_DIS
LIN {X -0.018,Y -185.902,Z 456.736,A 0.000,B 0.000,C 90.000,E1 132.405} C_DIS
LIN {X 0.042,Y -190.530,Z 456.722,A 0.000,B 0.000,C 90.000,E1 129.886} C_DIS
LIN {X 0.041,Y -194.713,Z 456.708,A 0.000,B 0.000,C 90.000,E1 127.443} C_DIS
LIN {X 0.031,Y -292.663,Z 456.708,A 0.000,B 0.000,C 90.000,E1 127.443} C_DIS
LIN {X -0.094,Y -294.161,Z 456.708,A 0.000,B 0.000,C 90.000,E1 127.443} C_DIS
LIN {X -0.063,Y -297.248,Z 456.707,A 0.000,B 0.000,C 90.000,E1 127.317} C_DIS
LIN {X -0.075,Y -300.594,Z 456.706,A 0.000,B 0.000,C 90.000,E1 127.076} C_DIS
LIN {X -0.013,Y -304.269,Z 456.703,A 0.000,B 0.000,C 90.000,E1 126.629} C_DIS
LIN {X 0.049,Y -306.175,Z 456.702,A 0.000,B 0.000,C 90.000,E1 126.297} C_DIS
LIN {X -0.137,Y -307.673,Z 456.700,A 0.000,B 0.000,C 90.000,E1 126.011} C_DIS
LIN {X 0.105,Y -309.881,Z 456.696,A 0.000,B 0.000,C 90.000,E1 125.311} C_DIS
LIN {X 0.067,Y -320.445,Z 456.678,A 0.000,B 0.000,C 90.000,E1 122.084} C_DIS
LIN {X 0.200,Y -331.314,Z 456.662,A 0.000,B 0.000,C 90.000,E1 119.205} C_DIS
LIN {X -0.003,Y -343.582,Z 456.647,A 0.000,B 0.000,C 90.000,E1 116.437} C_DIS
LIN {X -0.053,Y -355.745,Z 456.633,A 0.000,B 0.000,C 90.000,E1 114.003} C_DIS
LIN {X 0.090,Y -369.187,Z 456.620,A 0.000,B 0.000,C 90.000,E1 111.589} C_DIS
LIN {X -0.036,Y -384.003,Z 456.607,A 0.000,B 0.000,C 90.000,E1 109.268} C_DIS
LIN {X -0.041,Y -400.303,Z 456.594,A 0.000,B 0.000,C 90.000,E1 106.985} C_DIS
LIN {X -0.148,Y -418.208,Z 456.582,A 0.000,B 0.000,C 90.000,E1 104.773} C_DIS
LIN {X 0.050,Y -437.743,Z 456.570,A 0.000,B 0.000,C 90.000,E1 102.591} C_DIS
LIN {X 0.016,Y -458.064,Z 456.559,A 0.000,B 0.000,C 90.000,E1 100.602} C_DIS
LIN {X 0.014,Y -484.019,Z 456.546,A 0.000,B 0.000,C 90.000,E1 98.341} C_DIS
LIN {X 0.102,Y -485.975,Z 456.545,A 0.000,B 0.000,C 90.000,E1 98.106} C_DIS
LIN {X 0.188,Y -487.473,Z 456.544,A 0.000,B 0.000,C 90.000,E1 97.871} C_DIS
LIN {X 0.012,Y -488.731,Z 456.542,A 0.000,B 0.000,C 90.000,E1 97.644} C_DIS
LIN {X -0.099,Y -489.652,Z 456.541,A 0.000,B 0.000,C 90.000,E1 97.409} C_DIS
LIN {X 0.116,Y -490.650,Z 456.538,A 0.000,B 0.000,C 90.000,E1 96.891} C_DIS
LIN {X -0.150,Y -490.646,Z 456.536,A 0.000,B 0.000,C 90.000,E1 96.429} C_DIS
LIN {X 0.075,Y -489.641,Z 456.533,A 0.000,B 0.000,C 90.000,E1 95.910} C_DIS
LIN {X -0.081,Y -488.717,Z 456.532,A 0.000,B 0.000,C 90.000,E1 95.682} C_DIS
LIN {X -0.187,Y -487.456,Z 456.530,A 0.000,B 0.000,C 90.000,E1 95.448} C_DIS
LIN {X -0.018,Y -483.828,Z 456.527,A 0.000,B 0.000,C 90.000,E1 94.935} C_DIS
LIN {X -0.101,Y -465.828,Z 456.515,A 0.000,B 0.000,C 90.000,E1 92.694} C_DIS
LIN {X 0.024,Y -450.977,Z 456.504,A 0.000,B 0.000,C 90.000,E1 90.630} C_DIS
LIN {X 0.157,Y -434.228,Z 456.489,A 0.000,B 0.000,C 90.000,E1 87.993} C_DIS
LIN {X 0.142,Y -419.568,Z 456.476,A 0.000,B 0.000,C 90.000,E1 85.584} C_DIS
LIN {X 0.154,Y -407.019,Z 456.463,A 0.000,B 0.000,C 90.000,E1 83.394} C_DIS
LIN {X -0.071,Y -394.721,Z 456.451,A 0.000,B 0.000,C 90.000,E1 81.197} C_DIS
LIN {X -0.071,Y -382.374,Z 456.438,A 0.000,B 0.000,C 90.000,E1 78.926} C_DIS
LIN {X 0.065,Y -368.832,Z 456.424,A 0.000,B 0.000,C 90.000,E1 76.297} C_DIS
LIN {X 0.132,Y -357.483,Z 456.411,A 0.000,B 0.000,C 90.000,E1 73.921} C_DIS
LIN {X 0.092,Y -343.421,Z 456.392,A 0.000,B 0.000,C 90.000,E1 70.604} C_DIS
LIN {X -0.032,Y -331.746,Z 456.375,A 0.000,B 0.000,C 90.000,E1 67.539} C_DIS
LIN {X -0.077,Y -321.482,Z 456.359,A 0.000,B 0.000,C 90.000,E1 64.717} C_DIS
LIN {X -0.110,Y -313.730,Z 456.347,A 0.000,B 0.000,C 90.000,E1 62.487} C_DIS
LIN {X 0.013,Y -304.956,Z 456.333,A 0.000,B 0.000,C 90.000,E1 59.871} C_DIS
LIN {X 0.011,Y -294.514,Z 456.314,A 0.000,B 0.000,C 90.000,E1 56.580} C_DIS
LIN {X 0.089,Y -284.824,Z 456.296,A 0.000,B 0.000,C 90.000,E1 53.210} C_DIS
LIN {X 0.082,Y -279.167,Z 456.284,A 0.000,B 0.000,C 90.000,E1 51.170} C_DIS
LIN {X -0.063,Y -273.249,Z 456.273,A 0.000,B 0.000,C 90.000,E1 49.138} C_DIS
LIN {X 0.061,Y -267.117,Z 456.261,A 0.000,B 0.000,C 90.000,E1 47.025} C_DIS
LIN {X 0.041,Y -260.834,Z 456.250,A 0.000,B 0.000,C 90.000,E1 44.919} C_DIS
LIN {X 0.092,Y -254.414,Z 456.238,A 0.000,B 0.000,C 90.000,E1 42.771} C_DIS
LIN {X 0.037,Y -247.919,Z 456.226,A 0.000,B 0.000,C 90.000,E1 40.620} C_DIS
LIN {X 0.043,Y -237.368,Z 456.205,A 0.000,B 0.000,C 90.000,E1 36.950} C_DIS
LIN {X -0.087,Y -229.656,Z 456.189,A 0.000,B 0.000,C 90.000,E1 33.992} C_DIS
LIN {X 0.031,Y -222.610,Z 456.172,A 0.000,B 0.000,C 90.000,E1 30.924} C_DIS
LIN {X 0.016,Y -216.507,Z 456.155,A 0.000,B 0.000,C 90.000,E1 27.847} C_DIS
LIN {X -0.026,Y -209.983,Z 456.133,A 0.000,B 0.000,C 90.000,E1 23.951} C_DIS
LIN {X -0.034,Y -204.408,Z 456.111,A 0.000,B 0.000,C 90.000,E1 19.993} C_DIS
LIN {X 0.026,Y -199.862,Z 456.089,A 0.000,B 0.000,C 90.000,E1 15.969} C_DIS
LIN {X -0.041,Y -195.723,Z 456.062,A 0.000,B 0.000,C 90.000,E1 11.130} C_DIS
LIN {X 0.024,Y -192.483,Z 456.030,A 0.000,B 0.000,C 90.000,E1 5.391} C_DIS
LIN {X 0.093,Y -192.198,Z 455.965,A 0.000,B 0.000,C 90.000,E1 353.742} C_DIS
LIN {X -0.073,Y -195.195,Z 455.934,A 0.000,B 0.000,C 90.000,E1 348.049} C_DIS
LIN {X -0.001,Y -199.189,Z 455.906,A 0.000,B 0.000,C 90.000,E1 343.142} C_DIS
LIN {X 0.079,Y -203.525,Z 455.884,A 0.000,B 0.000,C 90.000,E1 339.082} C_DIS
LIN {X 0.021,Y -208.925,Z 455.862,A 0.000,B 0.000,C 90.000,E1 335.101} C_DIS
LIN {X -0.082,Y -215.143,Z 455.840,A 0.000,B 0.000,C 90.000,E1 331.179} C_DIS
LIN {X 0.052,Y -221.878,Z 455.818,A 0.000,B 0.000,C 90.000,E1 327.248} C_DIS
LIN {X 0.018,Y -229.265,Z 455.797,A 0.000,B 0.000,C 90.000,E1 323.417} C_DIS
LIN {X 0.075,Y -237.448,Z 455.776,A 0.000,B 0.000,C 90.000,E1 319.622} C_DIS
LIN {X 0.141,Y -246.716,Z 455.755,A 0.000,B 0.000,C 90.000,E1 315.891} C_DIS
LIN {X 0.162,Y -256.267,Z 455.737,A 0.000,B 0.000,C 90.000,E1 312.609} C_DIS
LIN {X 0.028,Y -268.260,Z 455.717,A 0.000,B 0.000,C 90.000,E1 309.072} C_DIS
LIN {X 0.036,Y -280.162,Z 455.700,A 0.000,B 0.000,C 90.000,E1 305.931} C_DIS
LIN {X -0.068,Y -294.223,Z 455.681,A 0.000,B 0.000,C 90.000,E1 302.546} C_DIS
LIN {X 0.027,Y -307.648,Z 455.664,A 0.000,B 0.000,C 90.000,E1 299.539} C_DIS
LIN {X 0.059,Y -322.313,Z 455.648,A 0.000,B 0.000,C 90.000,E1 296.616} C_DIS
LIN {X 0.078,Y -340.440,Z 455.630,A 0.000,B 0.000,C 90.000,E1 293.462} C_DIS
LIN {X -0.132,Y -356.644,Z 455.617,A 0.000,B 0.000,C 90.000,E1 291.046} C_DIS
LIN {X 0.100,Y -369.879,Z 455.607,A 0.000,B 0.000,C 90.000,E1 289.214} C_DIS
LIN {X 0.061,Y -393.764,Z 455.591,A 0.000,B 0.000,C 90.000,E1 286.315} C_DIS
LIN {X 0.010,Y -411.508,Z 455.580,A 0.000,B 0.000,C 90.000,E1 284.411} C_DIS
LIN {X 0.027,Y -426.905,Z 455.572,A 0.000,B 0.000,C 90.000,E1 282.883} C_DIS
LIN {X -0.061,Y -436.875,Z 455.566,A 0.000,B 0.000,C 90.000,E1 281.883} C_DIS
LIN {X 0.016,Y -446.584,Z 455.560,A 0.000,B 0.000,C 90.000,E1 280.838} C_DIS
LIN {X -0.167,Y -453.460,Z 455.556,A 0.000,B 0.000,C 90.000,E1 280.074} C_DIS
LIN {X -0.100,Y -461.962,Z 455.550,A 0.000,B 0.000,C 90.000,E1 279.029} C_DIS
LIN {X 0.234,Y -467.660,Z 455.546,A 0.000,B 0.000,C 90.000,E1 278.219} C_DIS
LIN {X 0.092,Y -472.755,Z 455.542,A 0.000,B 0.000,C 90.000,E1 277.473} C_DIS
LIN {X 0.062,Y -477.342,Z 455.537,A 0.000,B 0.000,C 90.000,E1 276.720} C_DIS
LIN {X 0.062,Y -481.489,Z 455.533,A 0.000,B 0.000,C 90.000,E1 275.967} C_DIS
LIN {X 0.051,Y -485.175,Z 455.529,A 0.000,B 0.000,C 90.000,E1 275.220} C_DIS
LIN {X 0.070,Y -488.151,Z 455.525,A 0.000,B 0.000,C 90.000,E1 274.473} C_DIS
LIN {X -0.221,Y -489.724,Z 455.522,A 0.000,B 0.000,C 90.000,E1 274.012} C_DIS
LIN {X -0.046,Y -490.810,Z 455.519,A 0.000,B 0.000,C 90.000,E1 273.498} C_DIS
LIN {X 0.170,Y -491.558,Z 455.517,A 0.000,B 0.000,C 90.000,E1 272.980} C_DIS
LIN {X -0.125,Y -491.921,Z 455.514,A 0.000,B 0.000,C 90.000,E1 272.522} C_DIS
LIN {X 0.077,Y -491.830,Z 455.511,A 0.000,B 0.000,C 90.000,E1 272.007} C_DIS
LIN {X -0.193,Y -491.384,Z 455.508,A 0.000,B 0.000,C 90.000,E1 271.547} C_DIS
LIN {X 0.011,Y -490.503,Z 455.506,A 0.000,B 0.000,C 90.000,E1 271.031} C_DIS
LIN {X 0.214,Y -489.139,Z 455.503,A 0.000,B 0.000,C 90.000,E1 270.516} C_DIS
LIN {X -0.076,Y -487.223,Z 455.500,A 0.000,B 0.000,C 90.000,E1 270.057} C_DIS
LIN {X 0.113,Y -484.679,Z 455.498,A 0.000,B 0.000,C 90.000,E1 269.542} C_DIS
LIN {X -0.199,Y -481.404,Z 455.495,A 0.000,B 0.000,C 90.000,E1 269.083} C_DIS
LIN {X -0.047,Y -477.249,Z 455.492,A 0.000,B 0.000,C 90.000,E1 268.568} C_DIS
LIN {X 0.097,Y -471.940,Z 455.489,A 0.000,B 0.000,C 90.000,E1 268.051} C_DIS
LIN {X 0.067,Y -469.081,Z 455.488,A 0.000,B 0.000,C 90.000,E1 267.822} C_DIS
LIN {X -0.173,Y -462.750,Z 455.486,A 0.000,B 0.000,C 90.000,E1 267.421} C_DIS
LIN {X 0.094,Y -456.229,Z 455.484,A 0.000,B 0.000,C 90.000,E1 267.020} C_DIS
LIN {X -0.104,Y -449.400,Z 455.482,A 0.000,B 0.000,C 90.000,E1 266.731} C_DIS
LIN {X 0.075,Y -442.265,Z 455.480,A 0.000,B 0.000,C 90.000,E1 266.445} C_DIS
LIN {X -0.202,Y -434.713,Z 455.479,A 0.000,B 0.000,C 90.000,E1 266.274} C_DIS
LIN {X -0.070,Y -426.257,Z 455.478,A 0.000,B 0.000,C 90.000,E1 266.102} C_DIS
LIN {X -0.020,Y -415.611,Z 455.478,A 0.000,B 0.000,C 90.000,E1 265.988} C_DIS
LIN {X 0.159,Y -409.832,Z 455.478,A 0.000,B 0.000,C 90.000,E1 265.931} C_DIS
LIN {X 0.111,Y -404.547,Z 455.477,A 0.000,B 0.000,C 90.000,E1 265.927} C_DIS
LIN {X 0.015,Y -180.917,Z 455.477,A 0.000,B 0.000,C 90.000,E1 265.927} C_DIS
LIN {X -0.028,Y -180.874,Z 455.473,A 0.000,B 0.000,C 90.000,E1 265.065} C_DIS
LIN {X 0.028,Y -178.990,Z 455.444,A 0.000,B 0.000,C 90.000,E1 259.982} C_DIS
LIN {X 0.039,Y -177.976,Z 455.435,A 0.000,B 0.000,C 90.000,E1 258.285} C_DIS
LIN {X 0.010,Y -175.619,Z 455.411,A 0.000,B 0.000,C 90.000,E1 254.047} C_DIS
LIN {X 0.069,Y -172.341,Z 455.388,A 0.000,B 0.000,C 90.000,E1 249.752} C_DIS
LIN {X 0.049,Y -171.817,Z 455.383,A 0.000,B 0.000,C 90.000,E1 248.901} C_DIS
LIN {X 0.056,Y -170.284,Z 455.373,A 0.000,B 0.000,C 90.000,E1 247.177} C_DIS
LIN {X -0.009,Y -166.823,Z 455.349,A 0.000,B 0.000,C 90.000,E1 242.871} C_DIS
LIN {X -0.091,Y -162.805,Z 455.325,A 0.000,B 0.000,C 90.000,E1 238.535} C_DIS
LIN {X -0.026,Y -161.492,Z 455.315,A 0.000,B 0.000,C 90.000,E1 236.755} C_DIS
LIN {X 0.023,Y -157.489,Z 455.291,A 0.000,B 0.000,C 90.000,E1 232.316} C_DIS
LIN {X -0.039,Y -155.506,Z 455.276,A 0.000,B 0.000,C 90.000,E1 229.666} C_DIS
LIN {X 0.012,Y -151.809,Z 455.251,A 0.000,B 0.000,C 90.000,E1 225.162} C_DIS
LIN {X 0.025,Y -150.021,Z 455.236,A 0.000,B 0.000,C 90.000,E1 222.447} C_DIS
LIN {X 0.055,Y -146.843,Z 455.211,A 0.000,B 0.000,C 90.000,E1 217.890} C_DIS
LIN {X -0.043,Y -145.426,Z 455.195,A 0.000,B 0.000,C 90.000,E1 215.185} C_DIS
LIN {X -0.047,Y -142.850,Z 455.170,A 0.000,B 0.000,C 90.000,E1 210.590} C_DIS
LIN {X 0.006,Y -141.466,Z 455.149,A 0.000,B 0.000,C 90.000,E1 206.873} C_DIS
LIN {X -0.003,Y -139.377,Z 455.113,A 0.000,B 0.000,C 90.000,E1 200.375} C_DIS
LIN {X -0.013,Y -138.828,Z 455.098,A 0.000,B 0.000,C 90.000,E1 197.583} C_DIS
LIN {X 0.051,Y -138.353,Z 455.056,A 0.000,B 0.000,C 90.000,E1 190.084} C_DIS
LIN {X 0.049,Y -139.528,Z 455.004,A 0.000,B 0.000,C 90.000,E1 180.745} C_DIS
LIN {X 0.003,Y -141.204,Z 454.973,A 0.000,B 0.000,C 90.000,E1 175.179} C_DIS
LIN {X -0.039,Y -142.579,Z 454.958,A 0.000,B 0.000,C 90.000,E1 172.413} C_DIS
LIN {X 0.058,Y -144.874,Z 454.932,A 0.000,B 0.000,C 90.000,E1 167.757} C_DIS
LIN {X 0.011,Y -147.500,Z 454.912,A 0.000,B 0.000,C 90.000,E1 164.102} C_DIS
LIN {X 0.087,Y -150.091,Z 454.891,A 0.000,B 0.000,C 90.000,E1 160.423} C_DIS
LIN {X -0.042,Y -153.445,Z 454.871,A 0.000,B 0.000,C 90.000,E1 156.847} C_DIS
LIN {X -0.048,Y -157.808,Z 454.846,A 0.000,B 0.000,C 90.000,E1 152.359} C_DIS
LIN {X -0.016,Y -162.089,Z 454.827,A 0.000,B 0.000,C 90.000,E1 148.791} C_DIS
LIN {X 0.008,Y -166.289,Z 454.807,A 0.000,B 0.000,C 90.000,E1 145.261} C_DIS
LIN {X 0.006,Y -171.306,Z 454.788,A 0.000,B 0.000,C 90.000,E1 141.778} C_DIS
LIN {X 0.040,Y -176.203,Z 454.769,A 0.000,B 0.000,C 90.000,E1 138.324} C_DIS
LIN {X -0.095,Y -180.479,Z 454.754,A 0.000,B 0.000,C 90.000,E1 135.810} C_DIS
LIN {X 0.017,Y -185.882,Z 454.736,A 0.000,B 0.000,C 90.000,E1 132.405} C_DIS
LIN {X -0.068,Y -190.509,Z 454.722,A 0.000,B 0.000,C 90.000,E1 129.930} C_DIS
LIN {X -0.001,Y -194.817,Z 454.708,A 0.000,B 0.000,C 90.000,E1 127.397} C_DIS
LIN {X 0.122,Y -293.288,Z 454.708,A 0.000,B 0.000,C 90.000,E1 127.363} C_DIS
LIN {X 0.013,Y -294.410,Z 454.708,A 0.000,B 0.000,C 90.000,E1 127.363} C_DIS
LIN {X 0.111,Y -298.561,Z 454.707,A 0.000,B 0.000,C 90.000,E1 127.156} C_DIS
LIN {X -0.029,Y -300.899,Z 454.706,A 0.000,B 0.000,C 90.000,E1 126.996} C_DIS
LIN {X 0.171,Y -304.104,Z 454.703,A 0.000,B 0.000,C 90.000,E1 126.583} C_DIS
LIN {X 0.003,Y -306.067,Z 454.702,A 0.000,B 0.000,C 90.000,E1 126.297} C_DIS
LIN {X 0.081,Y -307.605,Z 454.700,A 0.000,B 0.000,C 90.000,E1 125.964} C_DIS
LIN {X 0.042,Y -308.861,Z 454.698,A 0.000,B 0.000,C 90.000,E1 125.644} C_DIS
LIN {X 0.033,Y -320.445,Z 454.678,A 0.000,B 0.000,C 90.000,E1 122.084} C_DIS
LIN {X 0.166,Y -331.317,Z 454.662,A 0.000,B 0.000,C 90.000,E1 119.205} C_DIS
LIN {X -0.039,Y -343.586,Z 454.647,A 0.000,B 0.000,C 90.000,E1 116.437} C_DIS
LIN {X -0.090,Y -355.753,Z 454.633,A 0.000,B 0.000,C 90.000,E1 114.003} C_DIS
LIN {X 0.052,Y -369.197,Z 454.620,A 0.000,B 0.000,C 90.000,E1 111.589} C_DIS
LIN {X -0.075,Y -384.017,Z 454.607,A 0.000,B 0.000,C 90.000,E1 109.268} C_DIS
LIN {X -0.082,Y -400.321,Z 454.594,A 0.000,B 0.000,C 90.000,E1 106.985} C_DIS
LIN {X -0.190,Y -418.229,Z 454.582,A 0.000,B 0.000,C 90.000,E1 104.773} C_DIS
LIN {X 0.008,Y -437.767,Z 454.570,A 0.000,B 0.000,C 90.000,E1 102.591} C_DIS
LIN {X -0.026,Y -458.089,Z 454.559,A 0.000,B 0.000,C 90.000,E1 100.602} C_DIS
LIN {X -0.025,Y -484.071,Z 454.546,A 0.000,B 0.000,C 90.000,E1 98.341} C_DIS
LIN {X 0.074,Y -486.042,Z 454.545,A 0.000,B 0.000,C 90.000,E1 98.106} C_DIS
LIN {X 0.173,Y -487.555,Z 454.544,A 0.000,B 0.000,C 90.000,E1 97.871} C_DIS
LIN {X -0.002,Y -488.832,Z 454.542,A 0.000,B 0.000,C 90.000,E1 97.644} C_DIS
LIN {X -0.114,Y -489.772,Z 454.541,A 0.000,B 0.000,C 90.000,E1 97.409} C_DIS
LIN {X 0.101,Y -490.798,Z 454.538,A 0.000,B 0.000,C 90.000,E1 96.891} C_DIS
LIN {X -0.165,Y -490.822,Z 454.536,A 0.000,B 0.000,C 90.000,E1 96.429} C_DIS
LIN {X 0.061,Y -489.845,Z 454.533,A 0.000,B 0.000,C 90.000,E1 95.910} C_DIS
LIN {X -0.199,Y -487.696,Z 454.530,A 0.000,B 0.000,C 90.000,E1 95.448} C_DIS
LIN {X 0.130,Y -486.035,Z 454.529,A 0.000,B 0.000,C 90.000,E1 95.163} C_DIS
LIN {X -0.134,Y -476.053,Z 454.522,A 0.000,B 0.000,C 90.000,E1 93.955} C_DIS
LIN {X 0.017,Y -458.472,Z 454.509,A 0.000,B 0.000,C 90.000,E1 91.661} C_DIS
LIN {X 0.215,Y -446.055,Z 454.499,A 0.000,B 0.000,C 90.000,E1 89.828} C_DIS
LIN {X 0.171,Y -434.464,Z 454.489,A 0.000,B 0.000,C 90.000,E1 87.993} C_DIS
LIN {X 0.161,Y -419.771,Z 454.476,A 0.000,B 0.000,C 90.000,E1 85.584} C_DIS
LIN {X -0.169,Y -405.692,Z 454.462,A 0.000,B 0.000,C 90.000,E1 83.166} C_DIS
LIN {X -0.043,Y -394.962,Z 454.451,A 0.000,B 0.000,C 90.000,E1 81.197} C_DIS
LIN {X -0.037,Y -382.636,Z 454.438,A 0.000,B 0.000,C 90.000,E1 78.926} C_DIS
LIN {X 0.104,Y -369.112,Z 454.424,A 0.000,B 0.000,C 90.000,E1 76.297} C_DIS
LIN {X -0.168,Y -357.755,Z 454.411,A 0.000,B 0.000,C 90.000,E1 73.976} C_DIS
LIN {X 0.143,Y -343.656,Z 454.392,A 0.000,B 0.000,C 90.000,E1 70.604} C_DIS
LIN {X 0.024,Y -331.925,Z 454.375,A 0.000,B 0.000,C 90.000,E1 67.539} C_DIS
LIN {X -0.019,Y -321.612,Z 454.360,A 0.000,B 0.000,C 90.000,E1 64.717} C_DIS
LIN {X -0.050,Y -313.820,Z 454.347,A 0.000,B 0.000,C 90.000,E1 62.487} C_DIS
LIN {X 0.073,Y -305.020,Z 454.333,A 0.000,B 0.000,C 90.000,E1 59.871} C_DIS
LIN {X 0.070,Y -294.531,Z 454.314,A 0.000,B 0.000,C 90.000,E1 56.580} C_DIS
LIN {X -0.081,Y -284.824,Z 454.296,A 0.000,B 0.000,C 90.000,E1 53.256} C_DIS
LIN {X 0.140,Y -279.171,Z 454.284,A 0.000,B 0.000,C 90.000,E1 51.170} C_DIS
LIN {X -0.008,Y -273.279,Z 454.273,A 0.000,B 0.000,C 90.000,E1 49.138} C_DIS
LIN {X -0.079,Y -267.142,Z 454.261,A 0.000,B 0.000,C 90.000,E1 47.067} C_DIS
LIN {X 0.095,Y -260.871,Z 454.250,A 0.000,B 0.000,C 90.000,E1 44.919} C_DIS
LIN {X 0.145,Y -254.455,Z 454.238,A 0.000,B 0.000,C 90.000,E1 42.771} C_DIS
LIN {X 0.089,Y -247.963,Z 454.226,A 0.000,B 0.000,C 90.000,E1 40.620} C_DIS
LIN {X 0.095,Y -237.416,Z 454.205,A 0.000,B 0.000,C 90.000,E1 36.950} C_DIS
LIN {X -0.036,Y -229.689,Z 454.189,A 0.000,B 0.000,C 90.000,E1 33.992} C_DIS
LIN {X 0.083,Y -222.651,Z 454.172,A 0.000,B 0.000,C 90.000,E1 30.924} C_DIS
LIN {X 0.067,Y -216.555,Z 454.155,A 0.000,B 0.000,C 90.000,E1 27.847} C_DIS
LIN {X 0.024,Y -210.009,Z 454.133,A 0.000,B 0.000,C 90.000,E1 23.951} C_DIS
LIN {X 0.016,Y -204.415,Z 454.111,A 0.000,B 0.000,C 90.000,E1 19.993} C_DIS
LIN {X 0.074,Y -199.855,Z 454.089,A 0.000,B 0.000,C 90.000,E1 15.969} C_DIS
LIN {X 0.006,Y -195.679,Z 454.062,A 0.000,B 0.000,C 90.000,E1 11.130} C_DIS
LIN {X 0.068,Y -192.417,Z 454.030,A 0.000,B 0.000,C 90.000,E1 5.391} C_DIS
LIN {X 0.088,Y -192.075,Z 453.965,A 0.000,B 0.000,C 90.000,E1 353.742} C_DIS
LIN {X -0.083,Y -195.058,Z 453.933,A 0.000,B 0.000,C 90.000,E1 348.049} C_DIS
LIN {X -0.018,Y -199.034,Z 453.906,A 0.000,B 0.000,C 90.000,E1 343.142} C_DIS
LIN {X 0.056,Y -203.363,Z 453.884,A 0.000,B 0.000,C 90.000,E1 339.082} C_DIS
LIN {X -0.006,Y -208.775,Z 453.862,A 0.000,B 0.000,C 90.000,E1 335.101} C_DIS
LIN {X 0.073,Y -214.971,Z 453.840,A 0.000,B 0.000,C 90.000,E1 331.129} C_DIS
LIN {X 0.014,Y -221.710,Z 453.818,A 0.000,B 0.000,C 90.000,E1 327.248} C_DIS
LIN {X -0.028,Y -229.116,Z 453.797,A 0.000,B 0.000,C 90.000,E1 323.417} C_DIS
LIN {X 0.022,Y -237.311,Z 453.776,A 0.000,B 0.000,C 90.000,E1 319.622} C_DIS
LIN {X 0.082,Y -246.582,Z 453.755,A 0.000,B 0.000,C 90.000,E1 315.891} C_DIS
LIN {X 0.098,Y -256.153,Z 453.737,A 0.000,B 0.000,C 90.000,E1 312.609} C_DIS
LIN {X -0.042,Y -268.193,Z 453.717,A 0.000,B 0.000,C 90.000,E1 309.072} C_DIS
LIN {X -0.040,Y -280.123,Z 453.700,A 0.000,B 0.000,C 90.000,E1 305.931} C_DIS
LIN {X -0.149,Y -294.189,Z 453.681,A 0.000,B 0.000,C 90.000,E1 302.546} C_DIS
LIN {X -0.089,Y -306.102,Z 453.666,A 0.000,B 0.000,C 90.000,E1 299.873} C_DIS
LIN {X 0.046,Y -320.622,Z 453.650,A 0.000,B 0.000,C 90.000,E1 296.924} C_DIS
LIN {X 0.018,Y -336.701,Z 453.634,A 0.000,B 0.000,C 90.000,E1 294.079} C_DIS
LIN {X 0.124,Y -348.373,Z 453.623,A 0.000,B 0.000,C 90.000,E1 292.206} C_DIS
LIN {X -0.082,Y -363.157,Z 453.612,A 0.000,B 0.000,C 90.000,E1 290.120} C_DIS
LIN {X 0.024,Y -386.429,Z 453.595,A 0.000,B 0.000,C 90.000,E1 287.166} C_DIS
LIN {X -0.110,Y -401.442,Z 453.586,A 0.000,B 0.000,C 90.000,E1 285.481} C_DIS
LIN {X 0.173,Y -424.907,Z 453.573,A 0.000,B 0.000,C 90.000,E1 283.063} C_DIS
LIN {X 0.152,Y -434.903,Z 453.567,A 0.000,B 0.000,C 90.000,E1 282.063} C_DIS
LIN {X -0.019,Y -444.492,Z 453.562,A 0.000,B 0.000,C 90.000,E1 281.074} C_DIS
LIN {X -0.210,Y -451.522,Z 453.557,A 0.000,B 0.000,C 90.000,E1 280.310} C_DIS
LIN {X -0.165,Y -460.173,Z 453.551,A 0.000,B 0.000,C 90.000,E1 279.265} C_DIS
LIN {X 0.149,Y -466.069,Z 453.547,A 0.000,B 0.000,C 90.000,E1 278.454} C_DIS
LIN {X 0.062,Y -471.339,Z 453.543,A 0.000,B 0.000,C 90.000,E1 277.701} C_DIS
LIN {X 0.012,Y -476.088,Z 453.539,A 0.000,B 0.000,C 90.000,E1 276.947} C_DIS
LIN {X -0.189,Y -481.704,Z 453.533,A 0.000,B 0.000,C 90.000,E1 275.967} C_DIS
LIN {X -0.201,Y -485.390,Z 453.529,A 0.000,B 0.000,C 90.000,E1 275.220} C_DIS
LIN {X -0.181,Y -488.358,Z 453.525,A 0.000,B 0.000,C 90.000,E1 274.473} C_DIS
LIN {X 0.018,Y -489.873,Z 453.522,A 0.000,B 0.000,C 90.000,E1 273.955} C_DIS
LIN {X 0.195,Y -490.965,Z 453.519,A 0.000,B 0.000,C 90.000,E1 273.440} C_DIS
LIN {X -0.080,Y -491.666,Z 453.517,A 0.000,B 0.000,C 90.000,E1 272.980} C_DIS
LIN {X 0.117,Y -491.987,Z 453.514,A 0.000,B 0.000,C 90.000,E1 272.465} C_DIS
LIN {X -0.170,Y -491.900,Z 453.511,A 0.000,B 0.000,C 90.000,E1 272.007} C_DIS
LIN {X 0.051,Y -491.392,Z 453.508,A 0.000,B 0.000,C 90.000,E1 271.489} C_DIS
LIN {X -0.235,Y -490.471,Z 453.506,A 0.000,B 0.000,C 90.000,E1 271.031} C_DIS
LIN {X -0.032,Y -489.097,Z 453.503,A 0.000,B 0.000,C 90.000,E1 270.516} C_DIS
LIN {X 0.166,Y -487.151,Z 453.500,A 0.000,B 0.000,C 90.000,E1 270.000} C_DIS
LIN {X -0.131,Y -484.637,Z 453.497,A 0.000,B 0.000,C 90.000,E1 269.542} C_DIS
LIN {X 0.039,Y -481.303,Z 453.495,A 0.000,B 0.000,C 90.000,E1 269.026} C_DIS
LIN {X -0.125,Y -479.314,Z 453.493,A 0.000,B 0.000,C 90.000,E1 268.797} C_DIS
LIN {X 0.015,Y -474.535,Z 453.490,A 0.000,B 0.000,C 90.000,E1 268.282} C_DIS
LIN {X -0.148,Y -468.871,Z 453.488,A 0.000,B 0.000,C 90.000,E1 267.822} C_DIS
LIN {X 0.107,Y -462.565,Z 453.485,A 0.000,B 0.000,C 90.000,E1 267.364} C_DIS
LIN {X -0.055,Y -455.965,Z 453.483,A 0.000,B 0.000,C 90.000,E1 267.020} C_DIS
LIN {X -0.211,Y -449.109,Z 453.482,A 0.000,B 0.000,C 90.000,E1 266.731} C_DIS
LIN {X -0.015,Y -441.938,Z 453.480,A 0.000,B 0.000,C 90.000,E1 266.445} C_DIS
LIN {X 0.150,Y -434.253,Z 453.479,A 0.000,B 0.000,C 90.000,E1 266.216} C_DIS
LIN {X -0.136,Y -425.740,Z 453.478,A 0.000,B 0.000,C 90.000,E1 266.102} C_DIS
LIN {X -0.068,Y -414.354,Z 453.478,A 0.000,B 0.000,C 90.000,E1 265.988} C_DIS
LIN {X 0.148,Y -406.536,Z 453.477,A 0.000,B 0.000,C 90.000,E1 265.927} C_DIS
LIN {X 0.033,Y -180.918,Z 453.477,A 0.000,B 0.000,C 90.000,E1 265.927} C_DIS
LIN {X 0.066,Y -180.840,Z 453.472,A 0.000,B 0.000,C 90.000,E1 264.894} C_DIS
LIN {X -0.037,Y -178.882,Z 453.443,A 0.000,B 0.000,C 90.000,E1 259.690} C_DIS
LIN {X 0.038,Y -175.925,Z 453.414,A 0.000,B 0.000,C 90.000,E1 254.574} C_DIS
LIN {X -0.016,Y -175.362,Z 453.410,A 0.000,B 0.000,C 90.000,E1 253.740} C_DIS
LIN {X 0.042,Y -172.142,Z 453.386,A 0.000,B 0.000,C 90.000,E1 249.444} C_DIS
LIN {X 0.020,Y -171.605,Z 453.381,A 0.000,B 0.000,C 90.000,E1 248.592} C_DIS
LIN {X 0.008,Y -167.827,Z 453.357,A 0.000,B 0.000,C 90.000,E1 244.280} C_DIS
LIN {X 0.025,Y -166.553,Z 453.347,A 0.000,B 0.000,C 90.000,E1 242.538} C_DIS
LIN {X -0.065,Y -162.548,Z 453.323,A 0.000,B 0.000,C 90.000,E1 238.201} C_DIS
LIN {X -0.004,Y -161.226,Z 453.313,A 0.000,B 0.000,C 90.000,E1 236.421} C_DIS
LIN {X 0.031,Y -157.232,Z 453.289,A 0.000,B 0.000,C 90.000,E1 231.984} C_DIS
LIN {X 0.054,Y -155.957,Z 453.279,A 0.000,B 0.000,C 90.000,E1 230.194} C_DIS
LIN {X 0.012,Y -152.211,Z 453.254,A 0.000,B 0.000,C 90.000,E1 225.729} C_DIS
LIN {X 0.033,Y -150.455,Z 453.239,A 0.000,B 0.000,C 90.000,E1 223.014} C_DIS
LIN {X 0.059,Y -147.181,Z 453.214,A 0.000,B 0.000,C 90.000,E1 218.463} C_DIS
LIN {X 0.026,Y -145.198,Z 453.193,A 0.000,B 0.000,C 90.000,E1 214.818} C_DIS
LIN {X 0.060,Y -142.337,Z 453.163,A 0.000,B 0.000,C 90.000,E1 209.283} C_DIS
LIN {X -0.011,Y -141.725,Z 453.153,A 0.000,B 0.000,C 90.000,E1 207.462} C_DIS
LIN {X -0.028,Y -139.479,Z 453.116,A 0.000,B 0.000,C 90.000,E1 200.972} C_DIS
LIN {X -0.039,Y -138.977,Z 453.101,A 0.000,B 0.000,C 90.000,E1 198.181} C_DIS
LIN {X -0.054,Y -138.332,Z 453.054,A 0.000,B 0.000,C 90.000,E1 189.782} C_DIS
LIN {X -0.054,Y -139.430,Z 453.008,A 0.000,B 0.000,C 90.000,E1 181.375} C_DIS
LIN {X 0.000,Y -141.359,Z 452.971,A 0.000,B 0.000,C 90.000,E1 174.837} C_DIS
LIN {X -0.025,Y -142.712,Z 452.956,A 0.000,B 0.000,C 90.000,E1 172.064} C_DIS
LIN {X -0.066,Y -145.088,Z 452.930,A 0.000,B 0.000,C 90.000,E1 167.465} C_DIS
LIN {X 0.071,Y -147.713,Z 452.910,A 0.000,B 0.000,C 90.000,E1 163.740} C_DIS
LIN {X 0.012,Y -150.368,Z 452.890,A 0.000,B 0.000,C 90.000,E1 160.115} C_DIS
LIN {X 0.031,Y -153.795,Z 452.869,A 0.000,B 0.000,C 90.000,E1 156.485} C_DIS
LIN {X -0.050,Y -157.207,Z 452.849,A 0.000,B 0.000,C 90.000,E1 152.922} C_DIS
LIN {X 0.032,Y -161.371,Z 452.830,A 0.000,B 0.000,C 90.000,E1 149.331} C_DIS
LIN {X 0.043,Y -165.573,Z 452.810,A 0.000,B 0.000,C 90.000,E1 145.801} C_DIS
LIN {X -0.074,Y -170.492,Z 452.791,A 0.000,B 0.000,C 90.000,E1 142.351} C_DIS
LIN {X 0.075,Y -175.373,Z 452.772,A 0.000,B 0.000,C 90.000,E1 138.852} C_DIS
LIN {X -0.062,Y -180.997,Z 452.753,A 0.000,B 0.000,C 90.000,E1 135.486} C_DIS
LIN {X 0.062,Y -186.424,Z 452.734,A 0.000,B 0.000,C 90.000,E1 132.081} C_DIS
LIN {X 0.010,Y -191.052,Z 452.720,A 0.000,B 0.000,C 90.000,E1 129.600} C_DIS
LIN {X -0.082,Y -194.922,Z 452.707,A 0.000,B 0.000,C 90.000,E1 127.363} C_DIS
LIN {X 0.071,Y -293.285,Z 452.707,A 0.000,B 0.000,C 90.000,E1 127.317} C_DIS
LIN {X -0.129,Y -298.520,Z 452.706,A 0.000,B 0.000,C 90.000,E1 127.156} C_DIS
